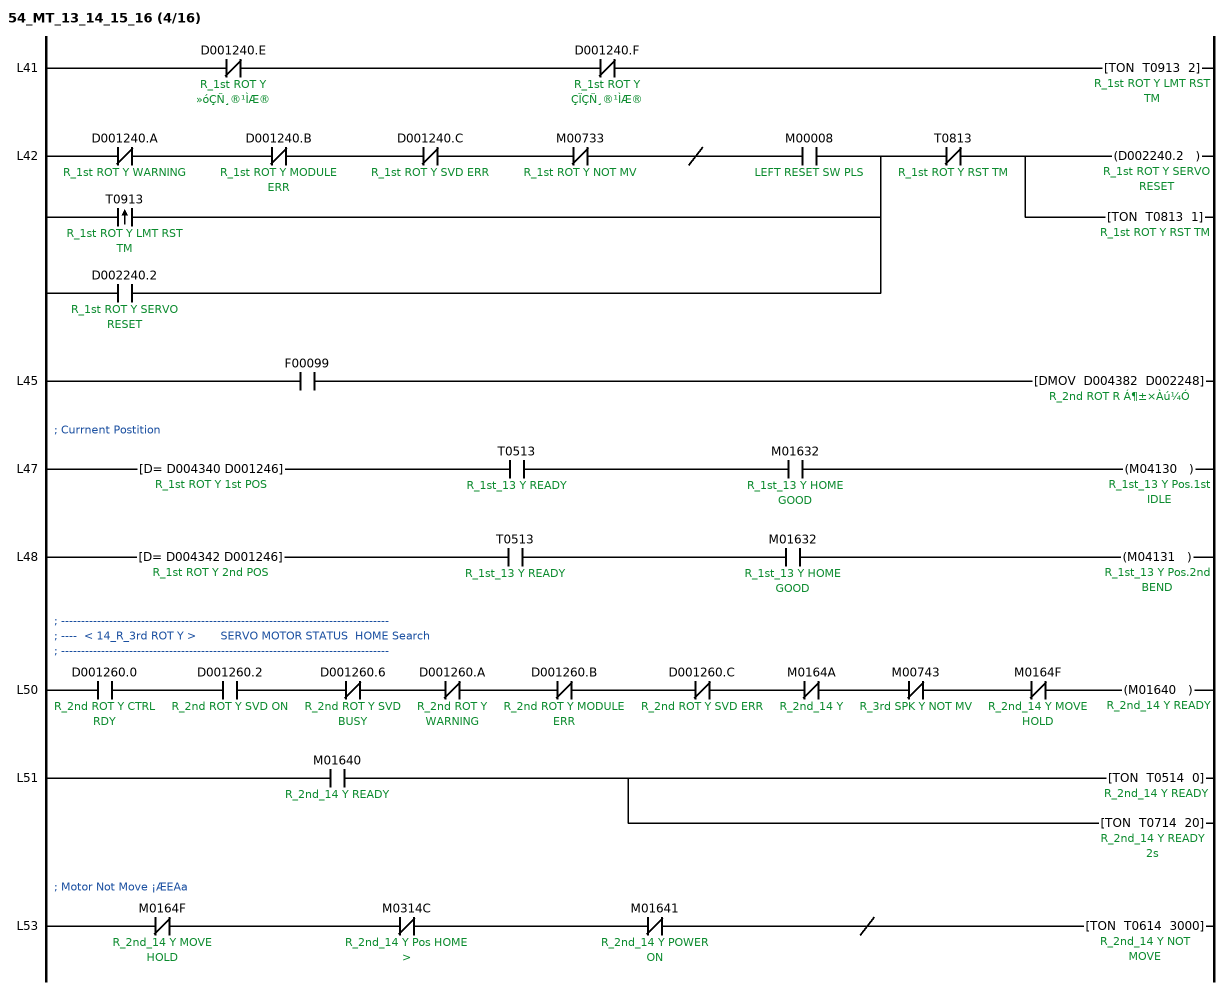
[picture p312: 54_MT_13_14_15_16 rungs L41-L53]
; L41
LOAD NOT  D001240.E	// R_1st ROT Y »óÇÑ¸®¹ÌÆ®
AND NOT   D001240.F	// R_1st ROT Y ÇÏÇÑ¸®¹ÌÆ®
TON       T0913 2	// R_1st ROT Y LMT RST TM
; L42
LOAD NOT  D001240.A	// R_1st ROT Y WARNING
AND NOT   D001240.B	// R_1st ROT Y MODULE ERR
AND NOT   D001240.C	// R_1st ROT Y SVD ERR
AND NOT   M00733	// R_1st ROT Y NOT MV
NOT
AND       M00008	// LEFT RESET SW PLS
ORP       T0913	// R_1st ROT Y LMT RST TM
OR        D002240.2	// R_1st ROT Y SERVO RESET
AND NOT   T0813	// R_1st ROT Y RST TM
OUT       D002240.2	// R_1st ROT Y SERVO RESET
TON       T0813 1	// R_1st ROT Y RST TM
; L45
LOAD      F00099
DMOV      D004382 D002248	// R_2nd ROT R Á¶±×Àú¼Ó
// Currnent Postition
; L47
LOADD=    D004340 D001246	// R_1st ROT Y 1st POS
AND       T0513	// R_1st_13 Y READY
AND       M01632	// R_1st_13 Y HOME GOOD
OUT       M04130	// R_1st_13 Y Pos.1st IDLE
; L48
LOADD=    D004342 D001246	// R_1st ROT Y 2nd POS
AND       T0513	// R_1st_13 Y READY
AND       M01632	// R_1st_13 Y HOME GOOD
OUT       M04131	// R_1st_13 Y Pos.2nd BEND
// ----------------------------------------------------------------------------------
// 
// ----  < 14_R_3rd ROT Y >       SERVO MOTOR STATUS  HOME Search
// 
// ----------------------------------------------------------------------------------
; L50
LOAD      D001260.0	// R_2nd ROT Y CTRL RDY
AND       D001260.2	// R_2nd ROT Y SVD ON
AND NOT   D001260.6	// R_2nd ROT Y SVD BUSY
AND NOT   D001260.A	// R_2nd ROT Y WARNING
AND NOT   D001260.B	// R_2nd ROT Y MODULE ERR
AND NOT   D001260.C	// R_2nd ROT Y SVD ERR
AND NOT   M0164A	// R_2nd_14 Y
AND NOT   M00743	// R_3rd SPK Y NOT MV
AND NOT   M0164F	// R_2nd_14 Y MOVE HOLD
OUT       M01640	// R_2nd_14 Y READY
; L51
LOAD      M01640	// R_2nd_14 Y READY
TON       T0514 0	// R_2nd_14 Y READY
TON       T0714 20	// R_2nd_14 Y READY 2s
; L53
LOAD NOT  M0164F	// R_2nd_14 Y MOVE HOLD
AND NOT   M0314C	// R_2nd_14 Y Pos HOME >
AND NOT   M01641	// R_2nd_14 Y POWER ON
NOT
TON       T0614 3000	// R_2nd_14 Y NOT MOVE
// output comment: Motor Not Move ¡ÆEAa

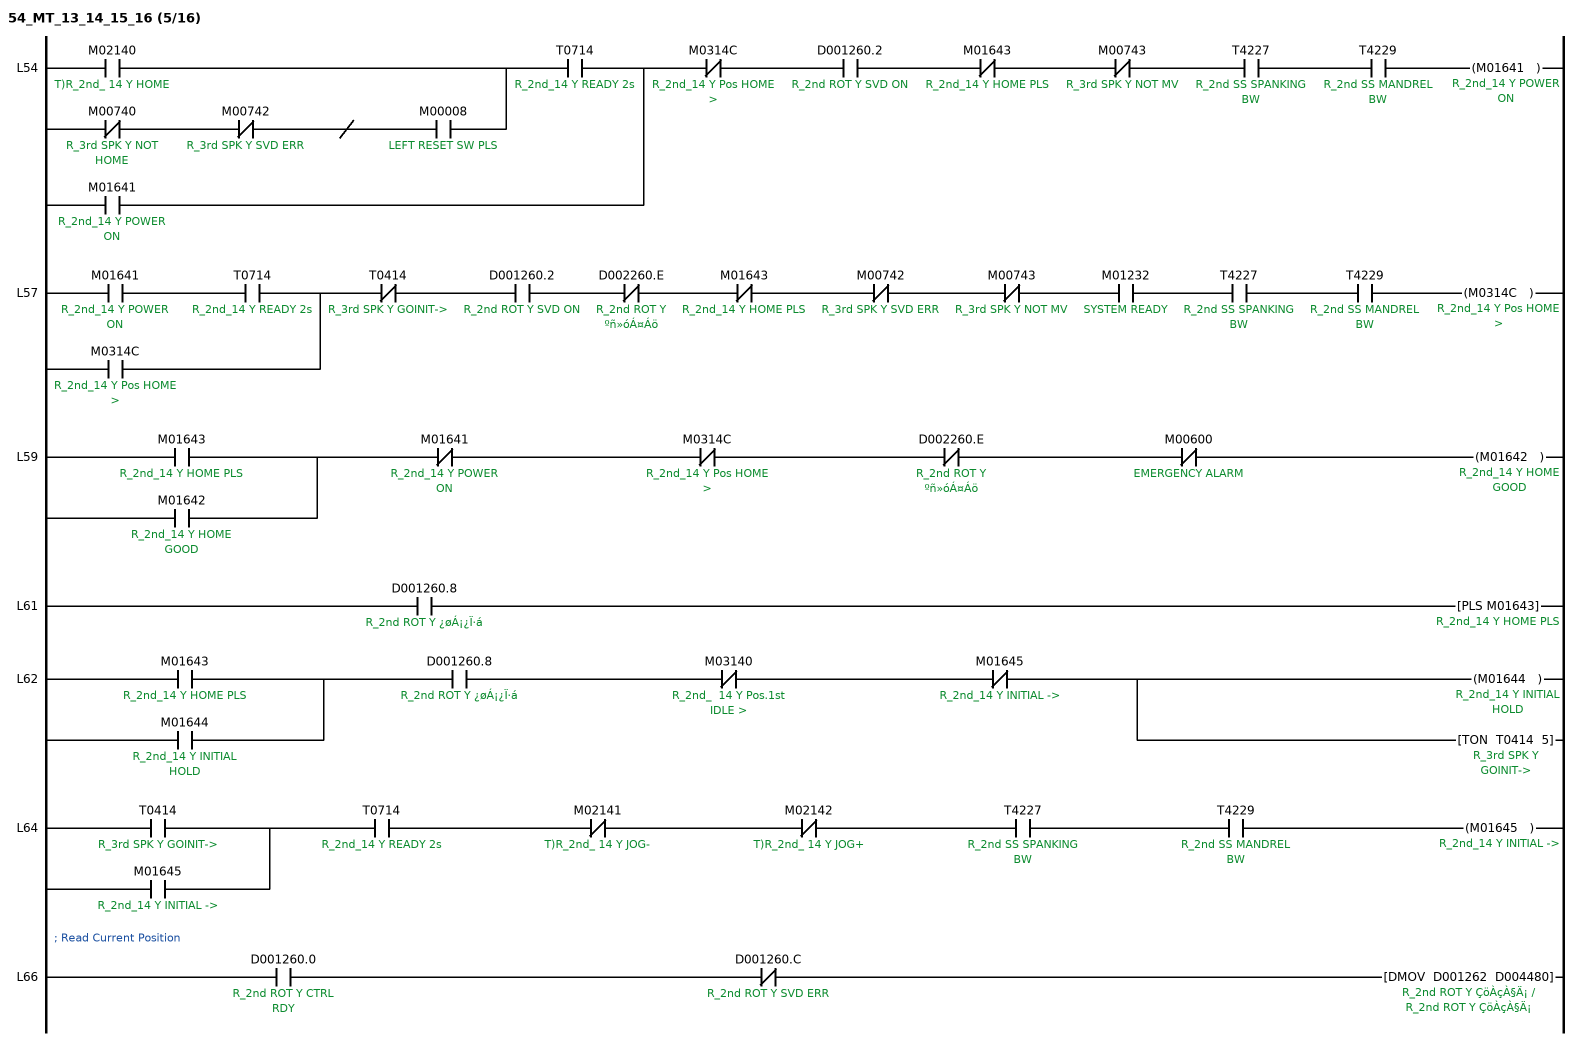
; L54
LOAD      M02140	// T)R_2nd_ 14 Y HOME
LOAD NOT  M00740	// R_3rd SPK Y NOT HOME
AND NOT   M00742	// R_3rd SPK Y SVD ERR
NOT
AND       M00008	// LEFT RESET SW PLS
OR LOAD
AND       T0714	// R_2nd_14 Y READY 2s
OR        M01641	// R_2nd_14 Y POWER ON
AND NOT   M0314C	// R_2nd_14 Y Pos HOME >
AND       D001260.2	// R_2nd ROT Y SVD ON
AND NOT   M01643	// R_2nd_14 Y HOME PLS
AND NOT   M00743	// R_3rd SPK Y NOT MV
AND       T4227	// R_2nd SS SPANKING BW
AND       T4229	// R_2nd SS MANDREL BW
OUT       M01641	// R_2nd_14 Y POWER ON
; L57
LOAD      M01641	// R_2nd_14 Y POWER ON
AND       T0714	// R_2nd_14 Y READY 2s
OR        M0314C	// R_2nd_14 Y Pos HOME >
AND NOT   T0414	// R_3rd SPK Y GOINIT->
AND       D001260.2	// R_2nd ROT Y SVD ON
AND NOT   D002260.E	// R_2nd ROT Y ºñ»óÁ¤Áö
AND NOT   M01643	// R_2nd_14 Y HOME PLS
AND NOT   M00742	// R_3rd SPK Y SVD ERR
AND NOT   M00743	// R_3rd SPK Y NOT MV
AND       M01232	// SYSTEM READY
AND       T4227	// R_2nd SS SPANKING BW
AND       T4229	// R_2nd SS MANDREL BW
OUT       M0314C	// R_2nd_14 Y Pos HOME >
; L59
LOAD      M01643	// R_2nd_14 Y HOME PLS
OR        M01642	// R_2nd_14 Y HOME GOOD
AND NOT   M01641	// R_2nd_14 Y POWER ON
AND NOT   M0314C	// R_2nd_14 Y Pos HOME >
AND NOT   D002260.E	// R_2nd ROT Y ºñ»óÁ¤Áö
AND NOT   M00600	// EMERGENCY ALARM
OUT       M01642	// R_2nd_14 Y HOME GOOD
; L61
LOAD      D001260.8	// R_2nd ROT Y ¿øÁ¡¿Ï·á
OUTP      M01643	// R_2nd_14 Y HOME PLS
; L62
LOAD      M01643	// R_2nd_14 Y HOME PLS
OR        M01644	// R_2nd_14 Y INITIAL HOLD
AND       D001260.8	// R_2nd ROT Y ¿øÁ¡¿Ï·á
AND NOT   M03140	// R_2nd_  14 Y Pos.1st IDLE >
AND NOT   M01645	// R_2nd_14 Y INITIAL ->
OUT       M01644	// R_2nd_14 Y INITIAL HOLD
TON       T0414 5	// R_3rd SPK Y GOINIT->
; L64
LOAD      T0414	// R_3rd SPK Y GOINIT->
OR        M01645	// R_2nd_14 Y INITIAL ->
AND       T0714	// R_2nd_14 Y READY 2s
AND NOT   M02141	// T)R_2nd_ 14 Y JOG-
AND NOT   M02142	// T)R_2nd_ 14 Y JOG+
AND       T4227	// R_2nd SS SPANKING BW
AND       T4229	// R_2nd SS MANDREL BW
OUT       M01645	// R_2nd_14 Y INITIAL ->
; L66
LOAD      D001260.0	// R_2nd ROT Y CTRL RDY
AND NOT   D001260.C	// R_2nd ROT Y SVD ERR
DMOV      D001262 D004480	// R_2nd ROT Y ÇöÀçÀ§Ä¡ / R_2nd ROT Y ÇöÀçÀ§Ä¡
// output comment: Read Current Position

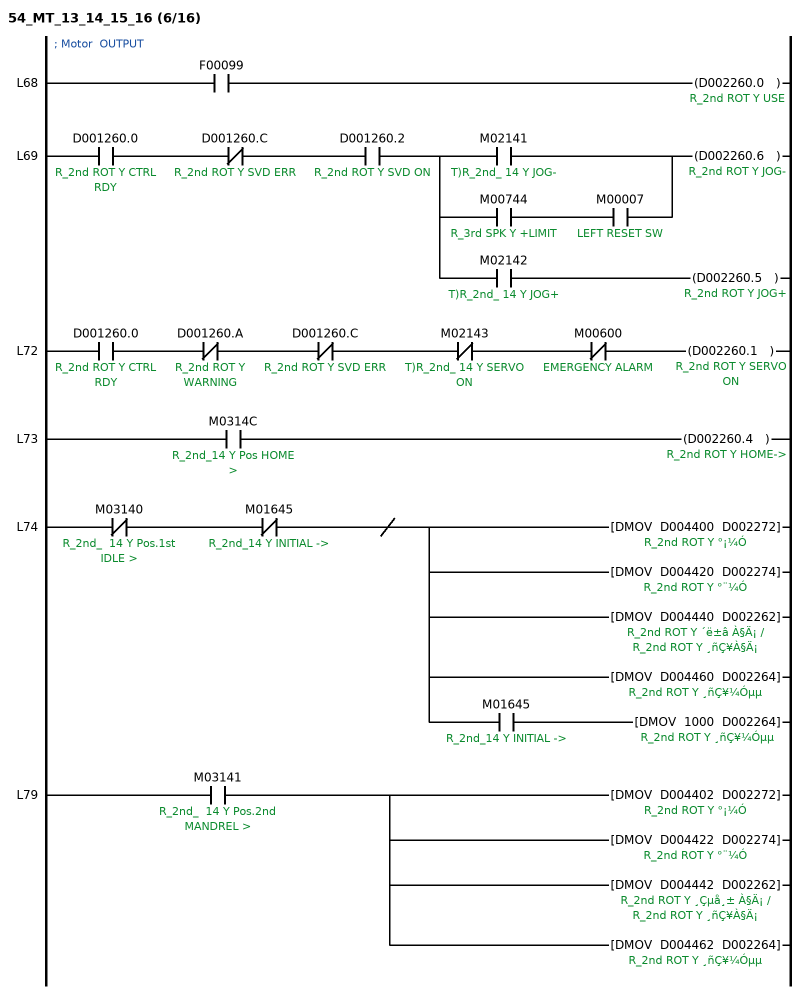
//  Motor  OUTPUT
; L68
LOAD      F00099
OUT       D002260.0	// R_2nd ROT Y USE
; L69
LOAD      D001260.0	// R_2nd ROT Y CTRL RDY
AND NOT   D001260.C	// R_2nd ROT Y SVD ERR
AND       D001260.2	// R_2nd ROT Y SVD ON
MPUSH
LOAD      M02141	// T)R_2nd_ 14 Y JOG-
LOAD      M00744	// R_3rd SPK Y +LIMIT
AND       M00007	// LEFT RESET SW
OR LOAD
AND LOAD
OUT       D002260.6	// R_2nd ROT Y JOG-
MPOP
AND       M02142	// T)R_2nd_ 14 Y JOG+
OUT       D002260.5	// R_2nd ROT Y JOG+
; L72
LOAD      D001260.0	// R_2nd ROT Y CTRL RDY
AND NOT   D001260.A	// R_2nd ROT Y WARNING
AND NOT   D001260.C	// R_2nd ROT Y SVD ERR
AND NOT   M02143	// T)R_2nd_ 14 Y SERVO ON
AND NOT   M00600	// EMERGENCY ALARM
OUT       D002260.1	// R_2nd ROT Y SERVO ON
; L73
LOAD      M0314C	// R_2nd_14 Y Pos HOME >
OUT       D002260.4	// R_2nd ROT Y HOME->
; L74
LOAD NOT  M03140	// R_2nd_  14 Y Pos.1st IDLE >
AND NOT   M01645	// R_2nd_14 Y INITIAL ->
NOT
DMOV      D004400 D002272	// R_2nd ROT Y °¡¼Ó
DMOV      D004420 D002274	// R_2nd ROT Y °¨¼Ó
DMOV      D004440 D002262	// R_2nd ROT Y ´ë±â À§Ä¡ / R_2nd ROT Y ¸ñÇ¥À§Ä¡
DMOV      D004460 D002264	// R_2nd ROT Y ¸ñÇ¥¼Óµµ
AND       M01645	// R_2nd_14 Y INITIAL ->
DMOV      1000 D002264	// R_2nd ROT Y ¸ñÇ¥¼Óµµ
; L79
LOAD      M03141	// R_2nd_  14 Y Pos.2nd MANDREL >
DMOV      D004402 D002272	// R_2nd ROT Y °¡¼Ó
DMOV      D004422 D002274	// R_2nd ROT Y °¨¼Ó
DMOV      D004442 D002262	// R_2nd ROT Y ¸Çµå¸± À§Ä¡ / R_2nd ROT Y ¸ñÇ¥À§Ä¡
DMOV      D004462 D002264	// R_2nd ROT Y ¸ñÇ¥¼Óµµ

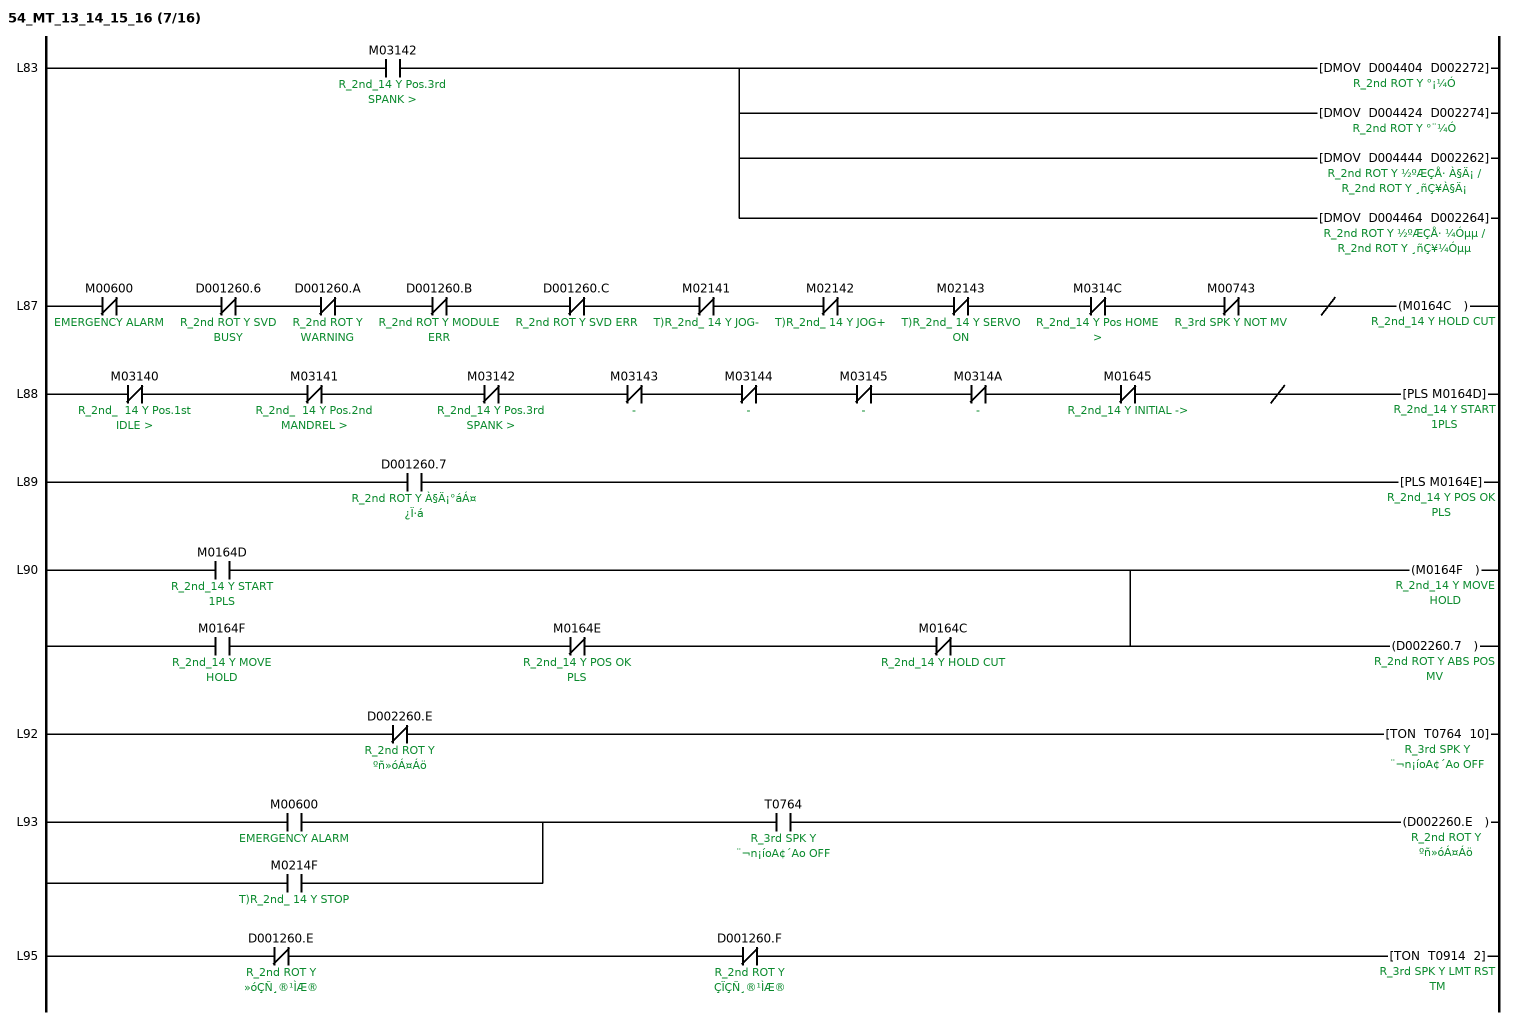
; L83
LOAD      M03142	// R_2nd_14 Y Pos.3rd SPANK >
DMOV      D004404 D002272	// R_2nd ROT Y °¡¼Ó
DMOV      D004424 D002274	// R_2nd ROT Y °¨¼Ó
DMOV      D004444 D002262	// R_2nd ROT Y ½ºÆÇÅ· À§Ä¡ / R_2nd ROT Y ¸ñÇ¥À§Ä¡
DMOV      D004464 D002264	// R_2nd ROT Y ½ºÆÇÅ· ¼Óµµ / R_2nd ROT Y ¸ñÇ¥¼Óµµ
; L87
LOAD NOT  M00600	// EMERGENCY ALARM
AND NOT   D001260.6	// R_2nd ROT Y SVD BUSY
AND NOT   D001260.A	// R_2nd ROT Y WARNING
AND NOT   D001260.B	// R_2nd ROT Y MODULE ERR
AND NOT   D001260.C	// R_2nd ROT Y SVD ERR
AND NOT   M02141	// T)R_2nd_ 14 Y JOG-
AND NOT   M02142	// T)R_2nd_ 14 Y JOG+
AND NOT   M02143	// T)R_2nd_ 14 Y SERVO ON
AND NOT   M0314C	// R_2nd_14 Y Pos HOME >
AND NOT   M00743	// R_3rd SPK Y NOT MV
NOT
OUT       M0164C	// R_2nd_14 Y HOLD CUT
; L88
LOAD NOT  M03140	// R_2nd_  14 Y Pos.1st IDLE >
AND NOT   M03141	// R_2nd_  14 Y Pos.2nd MANDREL >
AND NOT   M03142	// R_2nd_14 Y Pos.3rd SPANK >
AND NOT   M03143	// -
AND NOT   M03144	// -
AND NOT   M03145	// -
AND NOT   M0314A	// -
AND NOT   M01645	// R_2nd_14 Y INITIAL ->
NOT
OUTP      M0164D	// R_2nd_14 Y START 1PLS
; L89
LOAD      D001260.7	// R_2nd ROT Y À§Ä¡°áÁ¤ ¿Ï·á
OUTP      M0164E	// R_2nd_14 Y POS OK PLS
; L90
LOAD      M0164D	// R_2nd_14 Y START 1PLS
LOAD      M0164F	// R_2nd_14 Y MOVE HOLD
AND NOT   M0164E	// R_2nd_14 Y POS OK PLS
AND NOT   M0164C	// R_2nd_14 Y HOLD CUT
OR LOAD
OUT       M0164F	// R_2nd_14 Y MOVE HOLD
OUT       D002260.7	// R_2nd ROT Y ABS POS MV
; L92
LOAD NOT  D002260.E	// R_2nd ROT Y ºñ»óÁ¤Áö
TON       T0764 10	// R_3rd SPK Y ¨¬n¡íoA¢´Ao OFF
; L93
LOAD      M00600	// EMERGENCY ALARM
OR        M0214F	// T)R_2nd_ 14 Y STOP
AND       T0764	// R_3rd SPK Y ¨¬n¡íoA¢´Ao OFF
OUT       D002260.E	// R_2nd ROT Y ºñ»óÁ¤Áö
; L95
LOAD NOT  D001260.E	// R_2nd ROT Y »óÇÑ¸®¹ÌÆ®
AND NOT   D001260.F	// R_2nd ROT Y ÇÏÇÑ¸®¹ÌÆ®
TON       T0914 2	// R_3rd SPK Y LMT RST TM

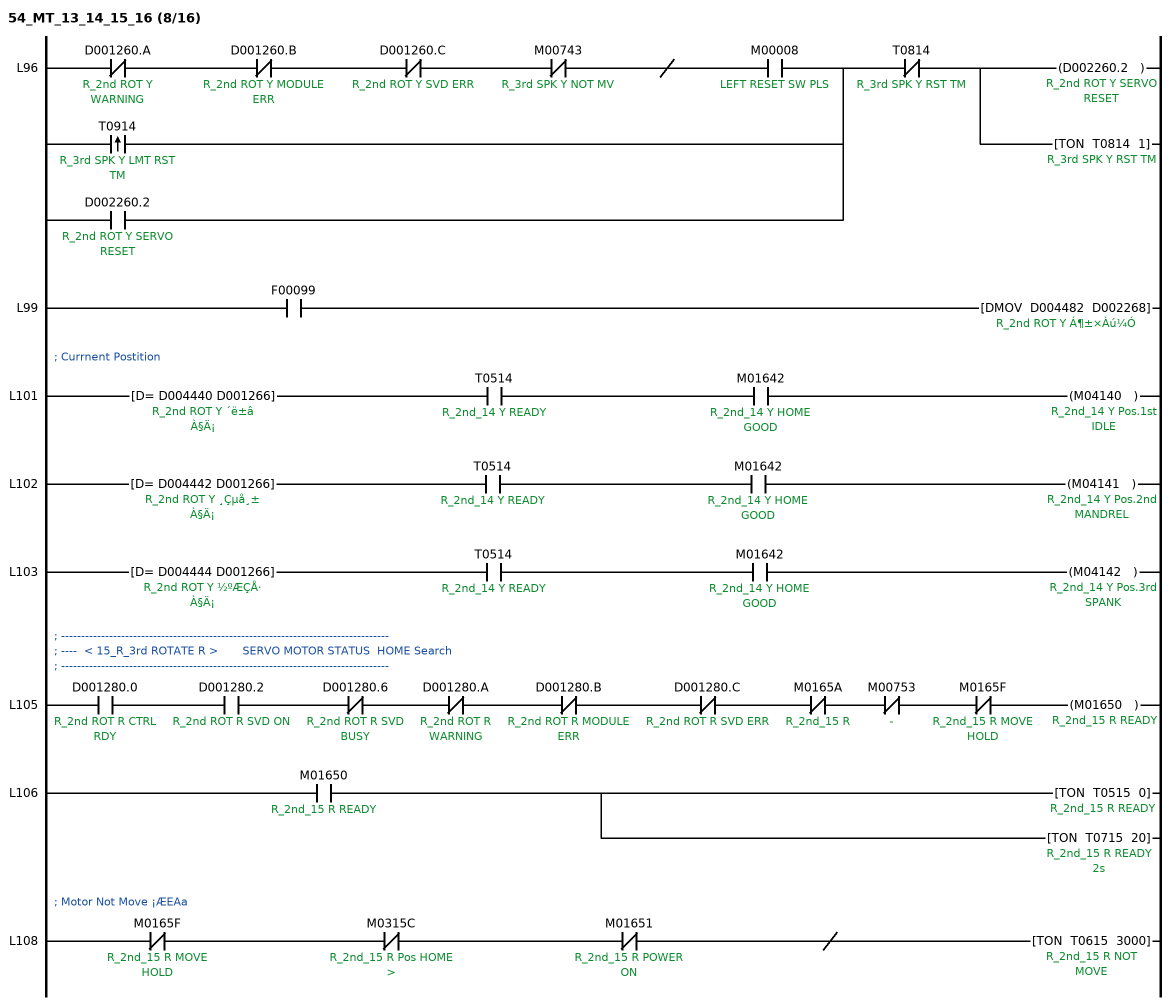
; L96
LOAD NOT  D001260.A	// R_2nd ROT Y WARNING
AND NOT   D001260.B	// R_2nd ROT Y MODULE ERR
AND NOT   D001260.C	// R_2nd ROT Y SVD ERR
AND NOT   M00743	// R_3rd SPK Y NOT MV
NOT
AND       M00008	// LEFT RESET SW PLS
ORP       T0914	// R_3rd SPK Y LMT RST TM
OR        D002260.2	// R_2nd ROT Y SERVO RESET
AND NOT   T0814	// R_3rd SPK Y RST TM
OUT       D002260.2	// R_2nd ROT Y SERVO RESET
TON       T0814 1	// R_3rd SPK Y RST TM
; L99
LOAD      F00099
DMOV      D004482 D002268	// R_2nd ROT Y Á¶±×Àú¼Ó
// Currnent Postition
; L101
LOADD=    D004440 D001266	// R_2nd ROT Y ´ë±â À§Ä¡
AND       T0514	// R_2nd_14 Y READY
AND       M01642	// R_2nd_14 Y HOME GOOD
OUT       M04140	// R_2nd_14 Y Pos.1st IDLE
; L102
LOADD=    D004442 D001266	// R_2nd ROT Y ¸Çµå¸± À§Ä¡
AND       T0514	// R_2nd_14 Y READY
AND       M01642	// R_2nd_14 Y HOME GOOD
OUT       M04141	// R_2nd_14 Y Pos.2nd MANDREL
; L103
LOADD=    D004444 D001266	// R_2nd ROT Y ½ºÆÇÅ· À§Ä¡
AND       T0514	// R_2nd_14 Y READY
AND       M01642	// R_2nd_14 Y HOME GOOD
OUT       M04142	// R_2nd_14 Y Pos.3rd SPANK
// ----------------------------------------------------------------------------------
// 
// ----  < 15_R_3rd ROTATE R >       SERVO MOTOR STATUS  HOME Search
// 
// ----------------------------------------------------------------------------------
; L105
LOAD      D001280.0	// R_2nd ROT R CTRL RDY
AND       D001280.2	// R_2nd ROT R SVD ON
AND NOT   D001280.6	// R_2nd ROT R SVD BUSY
AND NOT   D001280.A	// R_2nd ROT R WARNING
AND NOT   D001280.B	// R_2nd ROT R MODULE ERR
AND NOT   D001280.C	// R_2nd ROT R SVD ERR
AND NOT   M0165A	// R_2nd_15 R
AND NOT   M00753	// -
AND NOT   M0165F	// R_2nd_15 R MOVE HOLD
OUT       M01650	// R_2nd_15 R READY
; L106
LOAD      M01650	// R_2nd_15 R READY
TON       T0515 0	// R_2nd_15 R READY
TON       T0715 20	// R_2nd_15 R READY 2s
; L108
LOAD NOT  M0165F	// R_2nd_15 R MOVE HOLD
AND NOT   M0315C	// R_2nd_15 R Pos HOME >
AND NOT   M01651	// R_2nd_15 R POWER ON
NOT
TON       T0615 3000	// R_2nd_15 R NOT MOVE
// output comment: Motor Not Move ¡ÆEAa

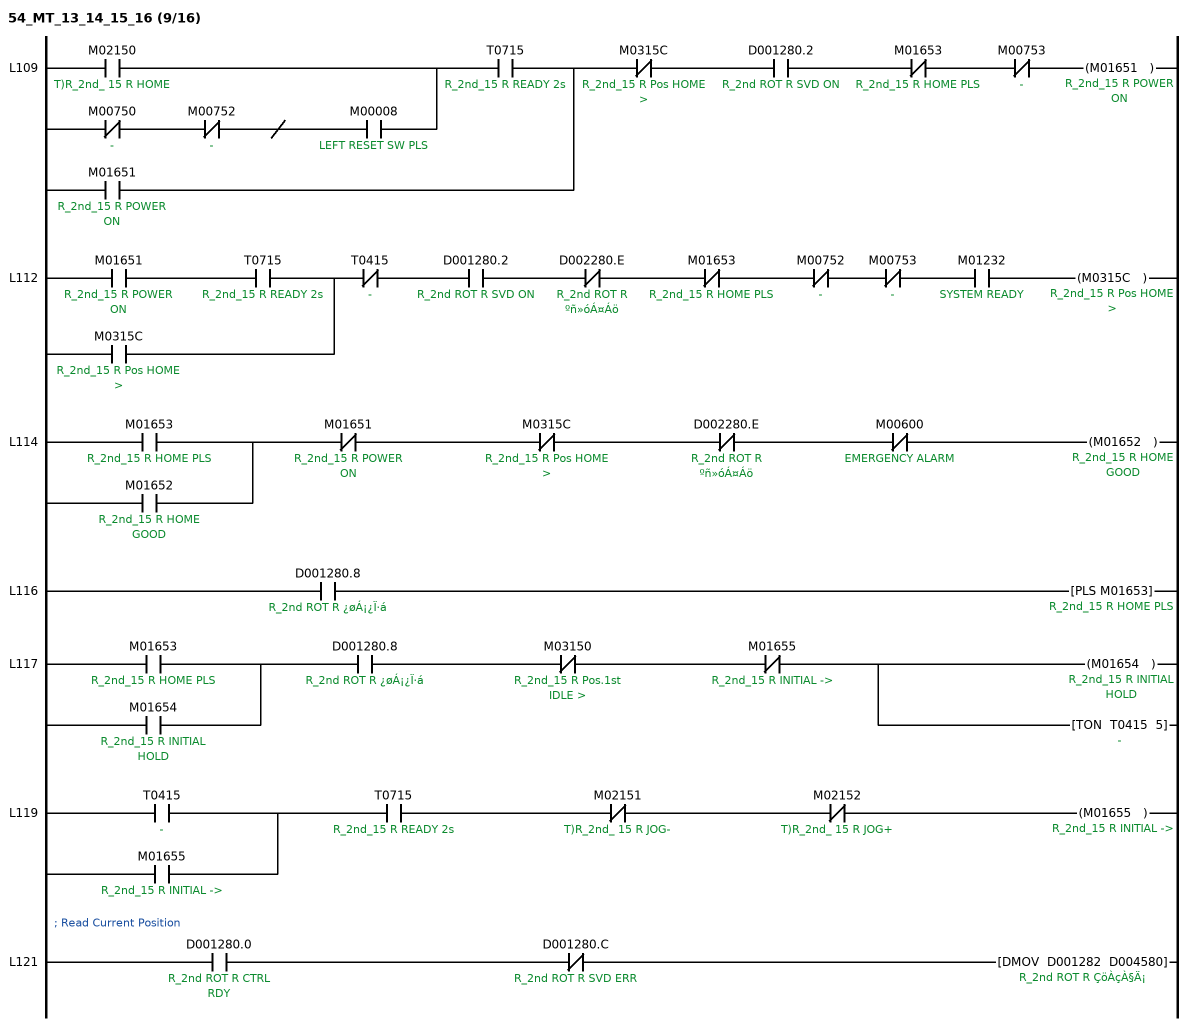
; L109
LOAD      M02150	// T)R_2nd_ 15 R HOME
LOAD NOT  M00750	// -
AND NOT   M00752	// -
NOT
AND       M00008	// LEFT RESET SW PLS
OR LOAD
AND       T0715	// R_2nd_15 R READY 2s
OR        M01651	// R_2nd_15 R POWER ON
AND NOT   M0315C	// R_2nd_15 R Pos HOME >
AND       D001280.2	// R_2nd ROT R SVD ON
AND NOT   M01653	// R_2nd_15 R HOME PLS
AND NOT   M00753	// -
OUT       M01651	// R_2nd_15 R POWER ON
; L112
LOAD      M01651	// R_2nd_15 R POWER ON
AND       T0715	// R_2nd_15 R READY 2s
OR        M0315C	// R_2nd_15 R Pos HOME >
AND NOT   T0415	// -
AND       D001280.2	// R_2nd ROT R SVD ON
AND NOT   D002280.E	// R_2nd ROT R ºñ»óÁ¤Áö
AND NOT   M01653	// R_2nd_15 R HOME PLS
AND NOT   M00752	// -
AND NOT   M00753	// -
AND       M01232	// SYSTEM READY
OUT       M0315C	// R_2nd_15 R Pos HOME >
; L114
LOAD      M01653	// R_2nd_15 R HOME PLS
OR        M01652	// R_2nd_15 R HOME GOOD
AND NOT   M01651	// R_2nd_15 R POWER ON
AND NOT   M0315C	// R_2nd_15 R Pos HOME >
AND NOT   D002280.E	// R_2nd ROT R ºñ»óÁ¤Áö
AND NOT   M00600	// EMERGENCY ALARM
OUT       M01652	// R_2nd_15 R HOME GOOD
; L116
LOAD      D001280.8	// R_2nd ROT R ¿øÁ¡¿Ï·á
OUTP      M01653	// R_2nd_15 R HOME PLS
; L117
LOAD      M01653	// R_2nd_15 R HOME PLS
OR        M01654	// R_2nd_15 R INITIAL HOLD
AND       D001280.8	// R_2nd ROT R ¿øÁ¡¿Ï·á
AND NOT   M03150	// R_2nd_15 R Pos.1st IDLE >
AND NOT   M01655	// R_2nd_15 R INITIAL ->
OUT       M01654	// R_2nd_15 R INITIAL HOLD
TON       T0415 5	// -
; L119
LOAD      T0415	// -
OR        M01655	// R_2nd_15 R INITIAL ->
AND       T0715	// R_2nd_15 R READY 2s
AND NOT   M02151	// T)R_2nd_ 15 R JOG-
AND NOT   M02152	// T)R_2nd_ 15 R JOG+
OUT       M01655	// R_2nd_15 R INITIAL ->
; L121
LOAD      D001280.0	// R_2nd ROT R CTRL RDY
AND NOT   D001280.C	// R_2nd ROT R SVD ERR
DMOV      D001282 D004580	// R_2nd ROT R ÇöÀçÀ§Ä¡
// output comment: Read Current Position

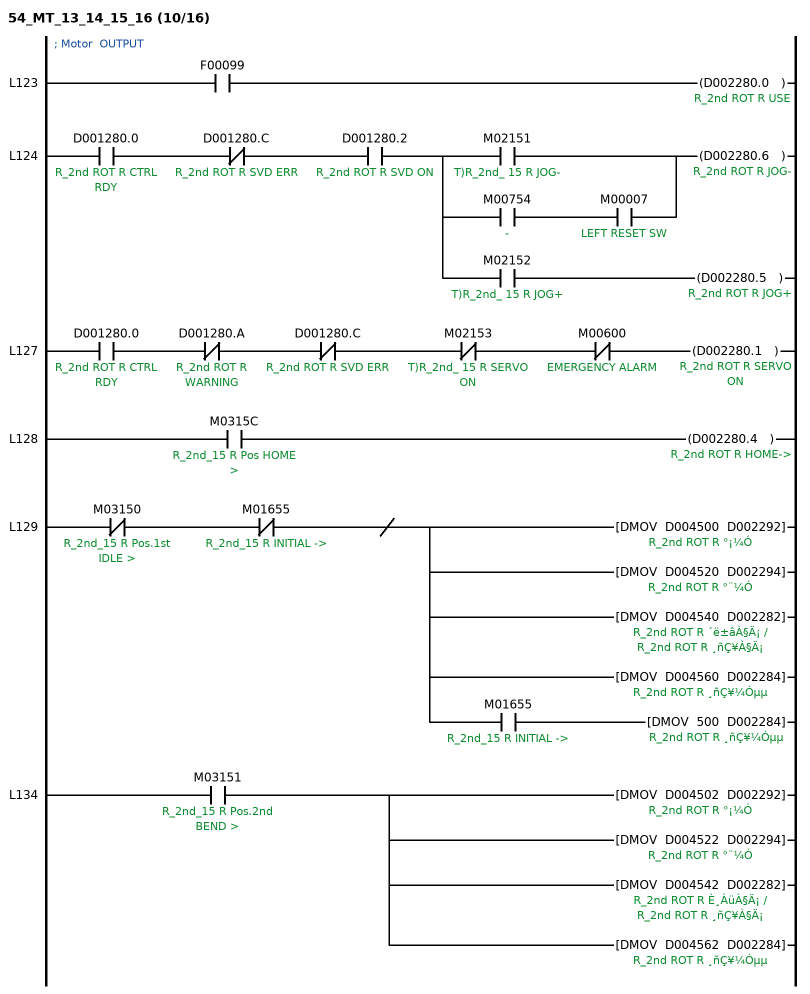
//  Motor  OUTPUT
; L123
LOAD      F00099
OUT       D002280.0	// R_2nd ROT R USE
; L124
LOAD      D001280.0	// R_2nd ROT R CTRL RDY
AND NOT   D001280.C	// R_2nd ROT R SVD ERR
AND       D001280.2	// R_2nd ROT R SVD ON
MPUSH
LOAD      M02151	// T)R_2nd_ 15 R JOG-
LOAD      M00754	// -
AND       M00007	// LEFT RESET SW
OR LOAD
AND LOAD
OUT       D002280.6	// R_2nd ROT R JOG-
MPOP
AND       M02152	// T)R_2nd_ 15 R JOG+
OUT       D002280.5	// R_2nd ROT R JOG+
; L127
LOAD      D001280.0	// R_2nd ROT R CTRL RDY
AND NOT   D001280.A	// R_2nd ROT R WARNING
AND NOT   D001280.C	// R_2nd ROT R SVD ERR
AND NOT   M02153	// T)R_2nd_ 15 R SERVO ON
AND NOT   M00600	// EMERGENCY ALARM
OUT       D002280.1	// R_2nd ROT R SERVO ON
; L128
LOAD      M0315C	// R_2nd_15 R Pos HOME >
OUT       D002280.4	// R_2nd ROT R HOME->
; L129
LOAD NOT  M03150	// R_2nd_15 R Pos.1st IDLE >
AND NOT   M01655	// R_2nd_15 R INITIAL ->
NOT
DMOV      D004500 D002292	// R_2nd ROT R °¡¼Ó
DMOV      D004520 D002294	// R_2nd ROT R °¨¼Ó
DMOV      D004540 D002282	// R_2nd ROT R ´ë±âÀ§Ä¡ / R_2nd ROT R ¸ñÇ¥À§Ä¡
DMOV      D004560 D002284	// R_2nd ROT R ¸ñÇ¥¼Óµµ
AND       M01655	// R_2nd_15 R INITIAL ->
DMOV      500 D002284	// R_2nd ROT R ¸ñÇ¥¼Óµµ
; L134
LOAD      M03151	// R_2nd_15 R Pos.2nd BEND >
DMOV      D004502 D002292	// R_2nd ROT R °¡¼Ó
DMOV      D004522 D002294	// R_2nd ROT R °¨¼Ó
DMOV      D004542 D002282	// R_2nd ROT R È¸ÀüÀ§Ä¡ / R_2nd ROT R ¸ñÇ¥À§Ä¡
DMOV      D004562 D002284	// R_2nd ROT R ¸ñÇ¥¼Óµµ

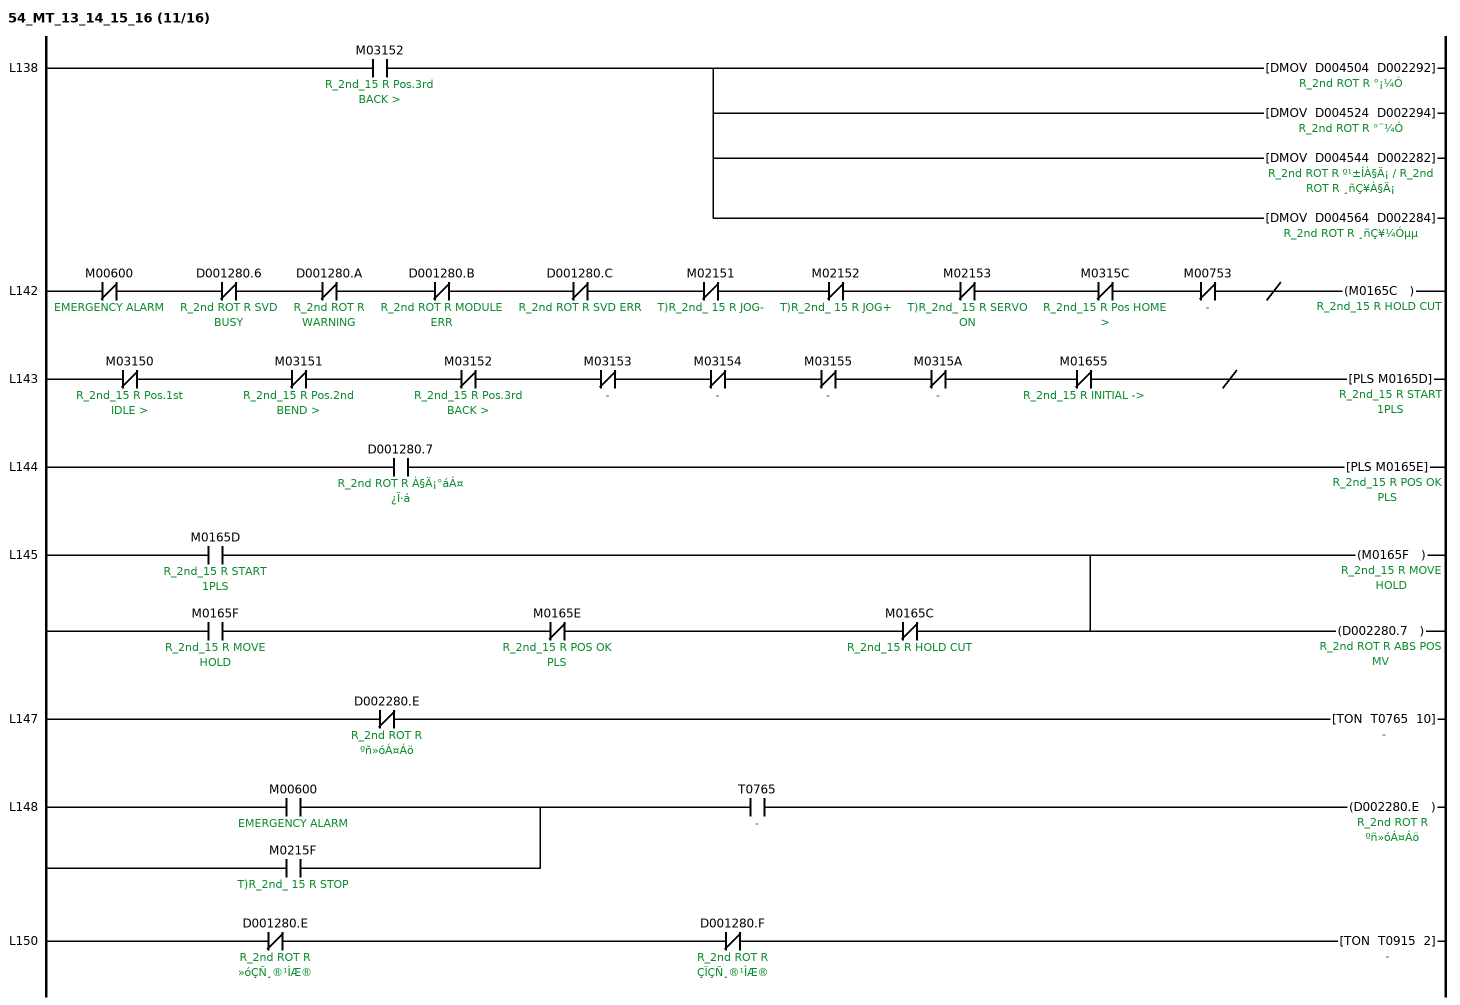
; L138
LOAD      M03152	// R_2nd_15 R Pos.3rd BACK >
DMOV      D004504 D002292	// R_2nd ROT R °¡¼Ó
DMOV      D004524 D002294	// R_2nd ROT R °¨¼Ó
DMOV      D004544 D002282	// R_2nd ROT R º¹±ÍÀ§Ä¡ / R_2nd ROT R ¸ñÇ¥À§Ä¡
DMOV      D004564 D002284	// R_2nd ROT R ¸ñÇ¥¼Óµµ
; L142
LOAD NOT  M00600	// EMERGENCY ALARM
AND NOT   D001280.6	// R_2nd ROT R SVD BUSY
AND NOT   D001280.A	// R_2nd ROT R WARNING
AND NOT   D001280.B	// R_2nd ROT R MODULE ERR
AND NOT   D001280.C	// R_2nd ROT R SVD ERR
AND NOT   M02151	// T)R_2nd_ 15 R JOG-
AND NOT   M02152	// T)R_2nd_ 15 R JOG+
AND NOT   M02153	// T)R_2nd_ 15 R SERVO ON
AND NOT   M0315C	// R_2nd_15 R Pos HOME >
AND NOT   M00753	// -
NOT
OUT       M0165C	// R_2nd_15 R HOLD CUT
; L143
LOAD NOT  M03150	// R_2nd_15 R Pos.1st IDLE >
AND NOT   M03151	// R_2nd_15 R Pos.2nd BEND >
AND NOT   M03152	// R_2nd_15 R Pos.3rd BACK >
AND NOT   M03153	// -
AND NOT   M03154	// -
AND NOT   M03155	// -
AND NOT   M0315A	// -
AND NOT   M01655	// R_2nd_15 R INITIAL ->
NOT
OUTP      M0165D	// R_2nd_15 R START 1PLS
; L144
LOAD      D001280.7	// R_2nd ROT R À§Ä¡°áÁ¤ ¿Ï·á
OUTP      M0165E	// R_2nd_15 R POS OK PLS
; L145
LOAD      M0165D	// R_2nd_15 R START 1PLS
LOAD      M0165F	// R_2nd_15 R MOVE HOLD
AND NOT   M0165E	// R_2nd_15 R POS OK PLS
AND NOT   M0165C	// R_2nd_15 R HOLD CUT
OR LOAD
OUT       M0165F	// R_2nd_15 R MOVE HOLD
OUT       D002280.7	// R_2nd ROT R ABS POS MV
; L147
LOAD NOT  D002280.E	// R_2nd ROT R ºñ»óÁ¤Áö
TON       T0765 10	// -
; L148
LOAD      M00600	// EMERGENCY ALARM
OR        M0215F	// T)R_2nd_ 15 R STOP
AND       T0765	// -
OUT       D002280.E	// R_2nd ROT R ºñ»óÁ¤Áö
; L150
LOAD NOT  D001280.E	// R_2nd ROT R »óÇÑ¸®¹ÌÆ®
AND NOT   D001280.F	// R_2nd ROT R ÇÏÇÑ¸®¹ÌÆ®
TON       T0915 2	// -

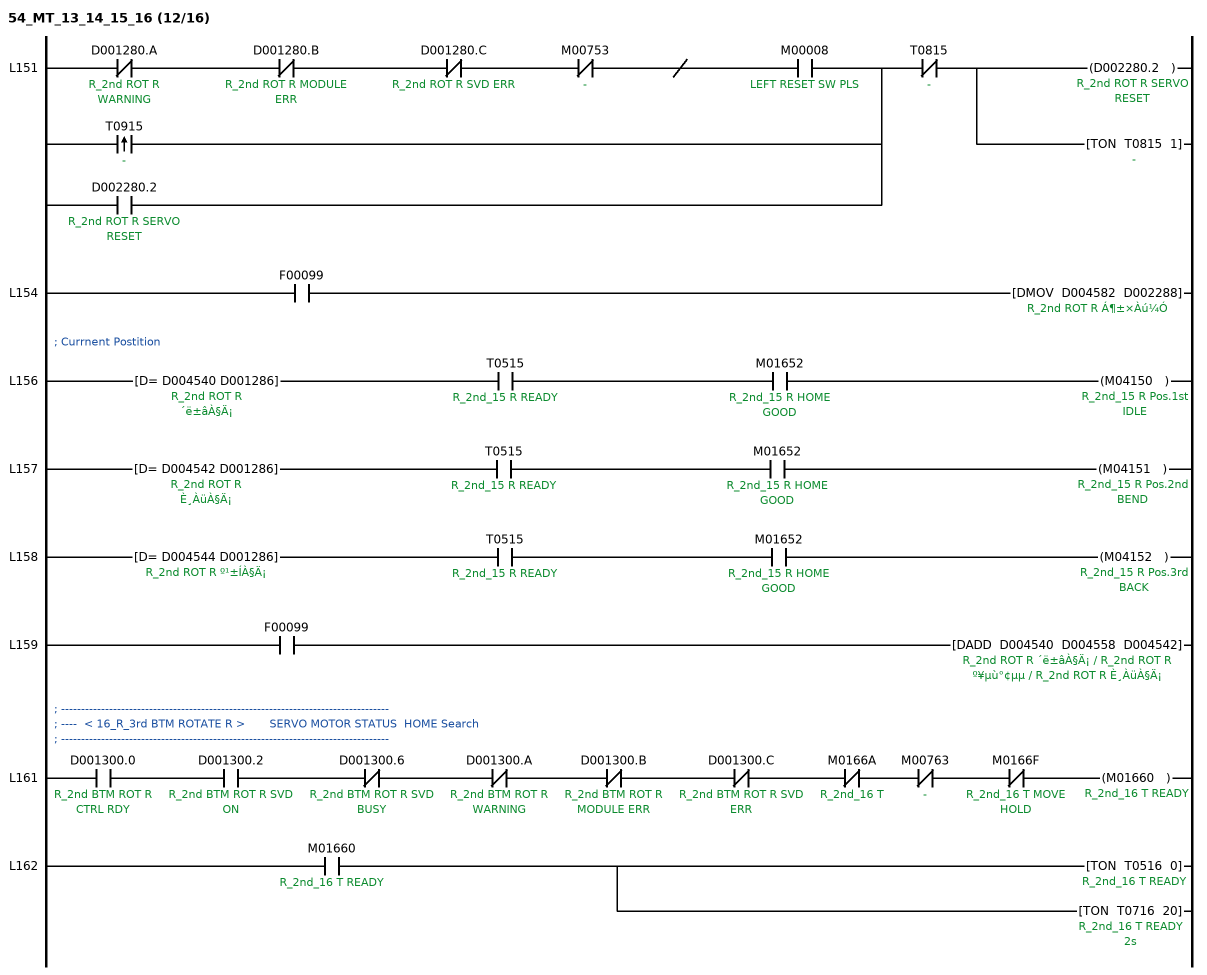
; L151
LOAD NOT  D001280.A	// R_2nd ROT R WARNING
AND NOT   D001280.B	// R_2nd ROT R MODULE ERR
AND NOT   D001280.C	// R_2nd ROT R SVD ERR
AND NOT   M00753	// -
NOT
AND       M00008	// LEFT RESET SW PLS
ORP       T0915	// -
OR        D002280.2	// R_2nd ROT R SERVO RESET
AND NOT   T0815	// -
OUT       D002280.2	// R_2nd ROT R SERVO RESET
TON       T0815 1	// -
; L154
LOAD      F00099
DMOV      D004582 D002288	// R_2nd ROT R Á¶±×Àú¼Ó
// Currnent Postition
; L156
LOADD=    D004540 D001286	// R_2nd ROT R ´ë±âÀ§Ä¡
AND       T0515	// R_2nd_15 R READY
AND       M01652	// R_2nd_15 R HOME GOOD
OUT       M04150	// R_2nd_15 R Pos.1st IDLE
; L157
LOADD=    D004542 D001286	// R_2nd ROT R È¸ÀüÀ§Ä¡
AND       T0515	// R_2nd_15 R READY
AND       M01652	// R_2nd_15 R HOME GOOD
OUT       M04151	// R_2nd_15 R Pos.2nd BEND
; L158
LOADD=    D004544 D001286	// R_2nd ROT R º¹±ÍÀ§Ä¡
AND       T0515	// R_2nd_15 R READY
AND       M01652	// R_2nd_15 R HOME GOOD
OUT       M04152	// R_2nd_15 R Pos.3rd BACK
; L159
LOAD      F00099
DADD      D004540 D004558 D004542	// R_2nd ROT R ´ë±âÀ§Ä¡ / R_2nd ROT R º¥µù°¢µµ / R_2nd ROT R È¸ÀüÀ§Ä¡
// ----------------------------------------------------------------------------------
// 
// ----  < 16_R_3rd BTM ROTATE R >       SERVO MOTOR STATUS  HOME Search
// 
// ----------------------------------------------------------------------------------
; L161
LOAD      D001300.0	// R_2nd BTM ROT R CTRL RDY
AND       D001300.2	// R_2nd BTM ROT R SVD ON
AND NOT   D001300.6	// R_2nd BTM ROT R SVD BUSY
AND NOT   D001300.A	// R_2nd BTM ROT R WARNING
AND NOT   D001300.B	// R_2nd BTM ROT R MODULE ERR
AND NOT   D001300.C	// R_2nd BTM ROT R SVD ERR
AND NOT   M0166A	// R_2nd_16 T
AND NOT   M00763	// -
AND NOT   M0166F	// R_2nd_16 T MOVE HOLD
OUT       M01660	// R_2nd_16 T READY
; L162
LOAD      M01660	// R_2nd_16 T READY
TON       T0516 0	// R_2nd_16 T READY
TON       T0716 20	// R_2nd_16 T READY 2s

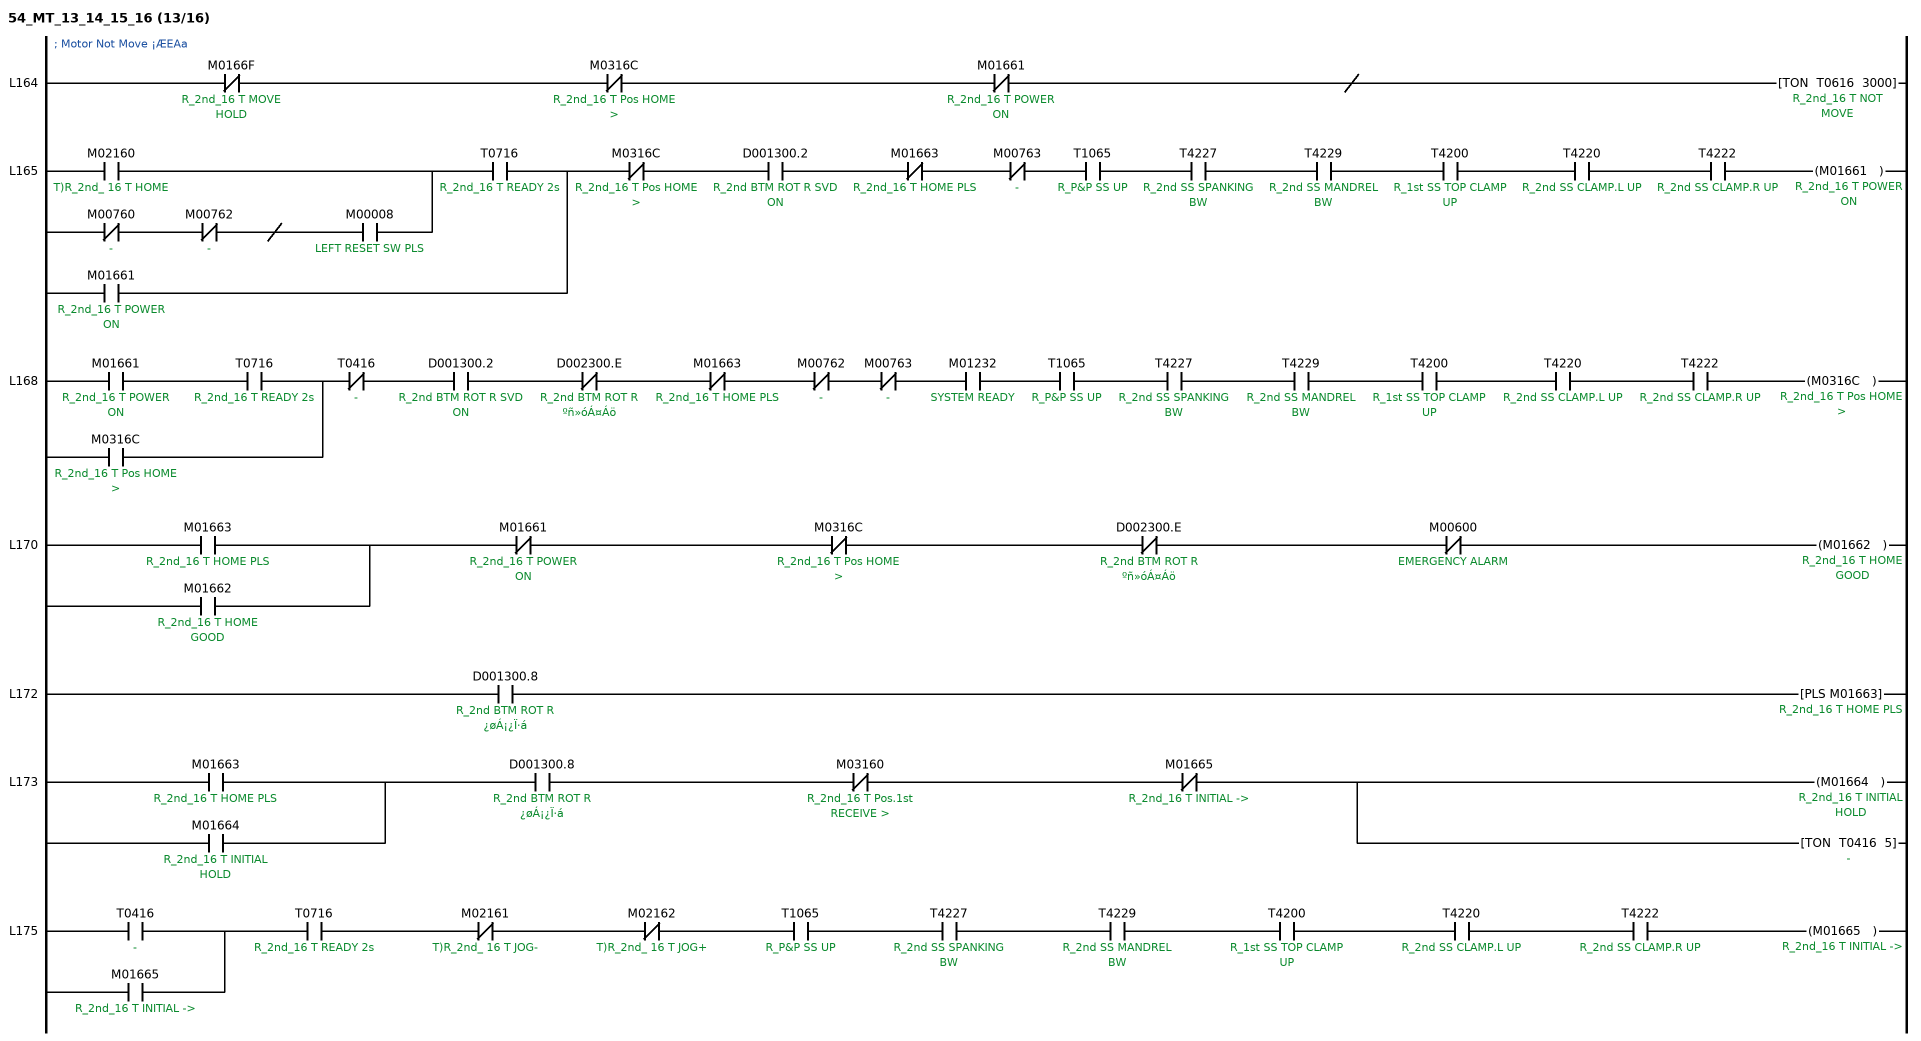
; L164
LOAD NOT  M0166F	// R_2nd_16 T MOVE HOLD
AND NOT   M0316C	// R_2nd_16 T Pos HOME >
AND NOT   M01661	// R_2nd_16 T POWER ON
NOT
TON       T0616 3000	// R_2nd_16 T NOT MOVE
// output comment: Motor Not Move ¡ÆEAa
; L165
LOAD      M02160	// T)R_2nd_ 16 T HOME
LOAD NOT  M00760	// -
AND NOT   M00762	// -
NOT
AND       M00008	// LEFT RESET SW PLS
OR LOAD
AND       T0716	// R_2nd_16 T READY 2s
OR        M01661	// R_2nd_16 T POWER ON
AND NOT   M0316C	// R_2nd_16 T Pos HOME >
AND       D001300.2	// R_2nd BTM ROT R SVD ON
AND NOT   M01663	// R_2nd_16 T HOME PLS
AND NOT   M00763	// -
AND       T1065	// R_P&P SS UP
AND       T4227	// R_2nd SS SPANKING BW
AND       T4229	// R_2nd SS MANDREL BW
AND       T4200	// R_1st SS TOP CLAMP UP
AND       T4220	// R_2nd SS CLAMP.L UP
AND       T4222	// R_2nd SS CLAMP.R UP
OUT       M01661	// R_2nd_16 T POWER ON
; L168
LOAD      M01661	// R_2nd_16 T POWER ON
AND       T0716	// R_2nd_16 T READY 2s
OR        M0316C	// R_2nd_16 T Pos HOME >
AND NOT   T0416	// -
AND       D001300.2	// R_2nd BTM ROT R SVD ON
AND NOT   D002300.E	// R_2nd BTM ROT R ºñ»óÁ¤Áö
AND NOT   M01663	// R_2nd_16 T HOME PLS
AND NOT   M00762	// -
AND NOT   M00763	// -
AND       M01232	// SYSTEM READY
AND       T1065	// R_P&P SS UP
AND       T4227	// R_2nd SS SPANKING BW
AND       T4229	// R_2nd SS MANDREL BW
AND       T4200	// R_1st SS TOP CLAMP UP
AND       T4220	// R_2nd SS CLAMP.L UP
AND       T4222	// R_2nd SS CLAMP.R UP
OUT       M0316C	// R_2nd_16 T Pos HOME >
; L170
LOAD      M01663	// R_2nd_16 T HOME PLS
OR        M01662	// R_2nd_16 T HOME GOOD
AND NOT   M01661	// R_2nd_16 T POWER ON
AND NOT   M0316C	// R_2nd_16 T Pos HOME >
AND NOT   D002300.E	// R_2nd BTM ROT R ºñ»óÁ¤Áö
AND NOT   M00600	// EMERGENCY ALARM
OUT       M01662	// R_2nd_16 T HOME GOOD
; L172
LOAD      D001300.8	// R_2nd BTM ROT R ¿øÁ¡¿Ï·á
OUTP      M01663	// R_2nd_16 T HOME PLS
; L173
LOAD      M01663	// R_2nd_16 T HOME PLS
OR        M01664	// R_2nd_16 T INITIAL HOLD
AND       D001300.8	// R_2nd BTM ROT R ¿øÁ¡¿Ï·á
AND NOT   M03160	// R_2nd_16 T Pos.1st RECEIVE >
AND NOT   M01665	// R_2nd_16 T INITIAL ->
OUT       M01664	// R_2nd_16 T INITIAL HOLD
TON       T0416 5	// -
; L175
LOAD      T0416	// -
OR        M01665	// R_2nd_16 T INITIAL ->
AND       T0716	// R_2nd_16 T READY 2s
AND NOT   M02161	// T)R_2nd_ 16 T JOG-
AND NOT   M02162	// T)R_2nd_ 16 T JOG+
AND       T1065	// R_P&P SS UP
AND       T4227	// R_2nd SS SPANKING BW
AND       T4229	// R_2nd SS MANDREL BW
AND       T4200	// R_1st SS TOP CLAMP UP
AND       T4220	// R_2nd SS CLAMP.L UP
AND       T4222	// R_2nd SS CLAMP.R UP
OUT       M01665	// R_2nd_16 T INITIAL ->

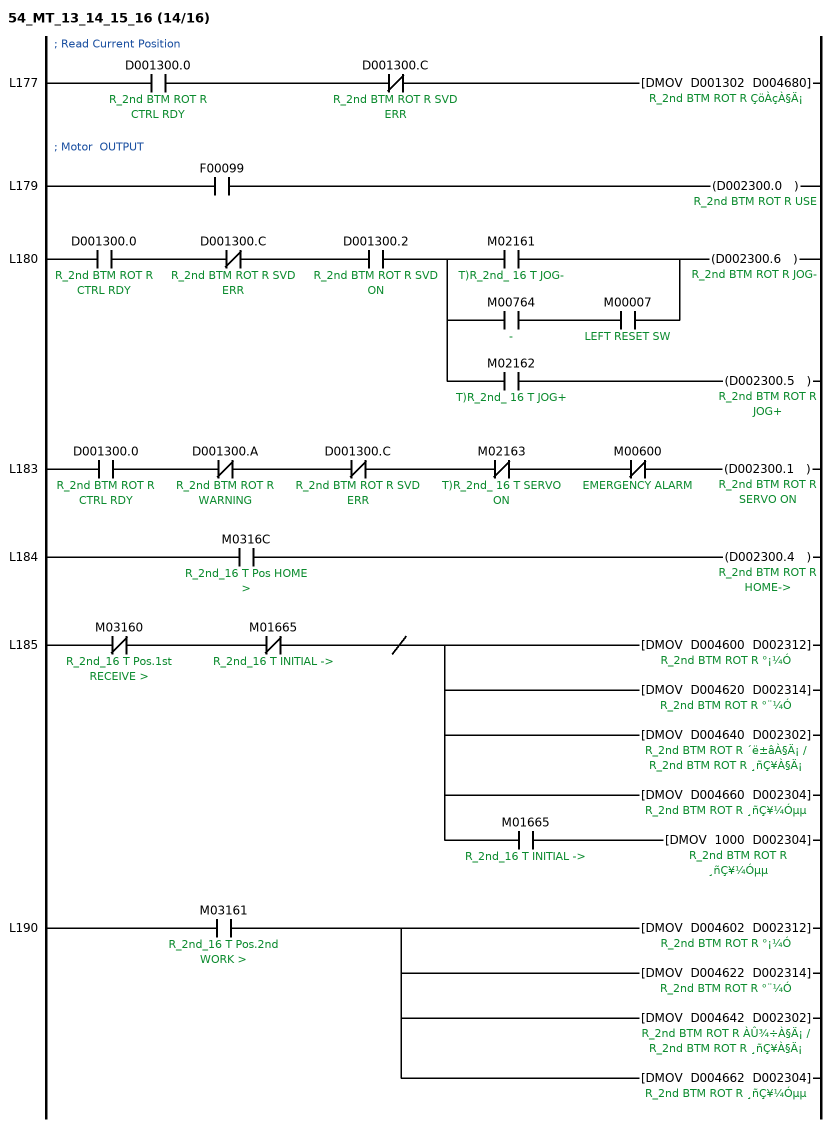
; L177
LOAD      D001300.0	// R_2nd BTM ROT R CTRL RDY
AND NOT   D001300.C	// R_2nd BTM ROT R SVD ERR
DMOV      D001302 D004680	// R_2nd BTM ROT R ÇöÀçÀ§Ä¡
// output comment: Read Current Position
//  Motor  OUTPUT
; L179
LOAD      F00099
OUT       D002300.0	// R_2nd BTM ROT R USE
; L180
LOAD      D001300.0	// R_2nd BTM ROT R CTRL RDY
AND NOT   D001300.C	// R_2nd BTM ROT R SVD ERR
AND       D001300.2	// R_2nd BTM ROT R SVD ON
MPUSH
LOAD      M02161	// T)R_2nd_ 16 T JOG-
LOAD      M00764	// -
AND       M00007	// LEFT RESET SW
OR LOAD
AND LOAD
OUT       D002300.6	// R_2nd BTM ROT R JOG-
MPOP
AND       M02162	// T)R_2nd_ 16 T JOG+
OUT       D002300.5	// R_2nd BTM ROT R JOG+
; L183
LOAD      D001300.0	// R_2nd BTM ROT R CTRL RDY
AND NOT   D001300.A	// R_2nd BTM ROT R WARNING
AND NOT   D001300.C	// R_2nd BTM ROT R SVD ERR
AND NOT   M02163	// T)R_2nd_ 16 T SERVO ON
AND NOT   M00600	// EMERGENCY ALARM
OUT       D002300.1	// R_2nd BTM ROT R SERVO ON
; L184
LOAD      M0316C	// R_2nd_16 T Pos HOME >
OUT       D002300.4	// R_2nd BTM ROT R HOME->
; L185
LOAD NOT  M03160	// R_2nd_16 T Pos.1st RECEIVE >
AND NOT   M01665	// R_2nd_16 T INITIAL ->
NOT
DMOV      D004600 D002312	// R_2nd BTM ROT R °¡¼Ó
DMOV      D004620 D002314	// R_2nd BTM ROT R °¨¼Ó
DMOV      D004640 D002302	// R_2nd BTM ROT R ´ë±âÀ§Ä¡ / R_2nd BTM ROT R ¸ñÇ¥À§Ä¡
DMOV      D004660 D002304	// R_2nd BTM ROT R ¸ñÇ¥¼Óµµ
AND       M01665	// R_2nd_16 T INITIAL ->
DMOV      1000 D002304	// R_2nd BTM ROT R ¸ñÇ¥¼Óµµ
; L190
LOAD      M03161	// R_2nd_16 T Pos.2nd WORK >
DMOV      D004602 D002312	// R_2nd BTM ROT R °¡¼Ó
DMOV      D004622 D002314	// R_2nd BTM ROT R °¨¼Ó
DMOV      D004642 D002302	// R_2nd BTM ROT R ÀÛ¾÷À§Ä¡ / R_2nd BTM ROT R ¸ñÇ¥À§Ä¡
DMOV      D004662 D002304	// R_2nd BTM ROT R ¸ñÇ¥¼Óµµ

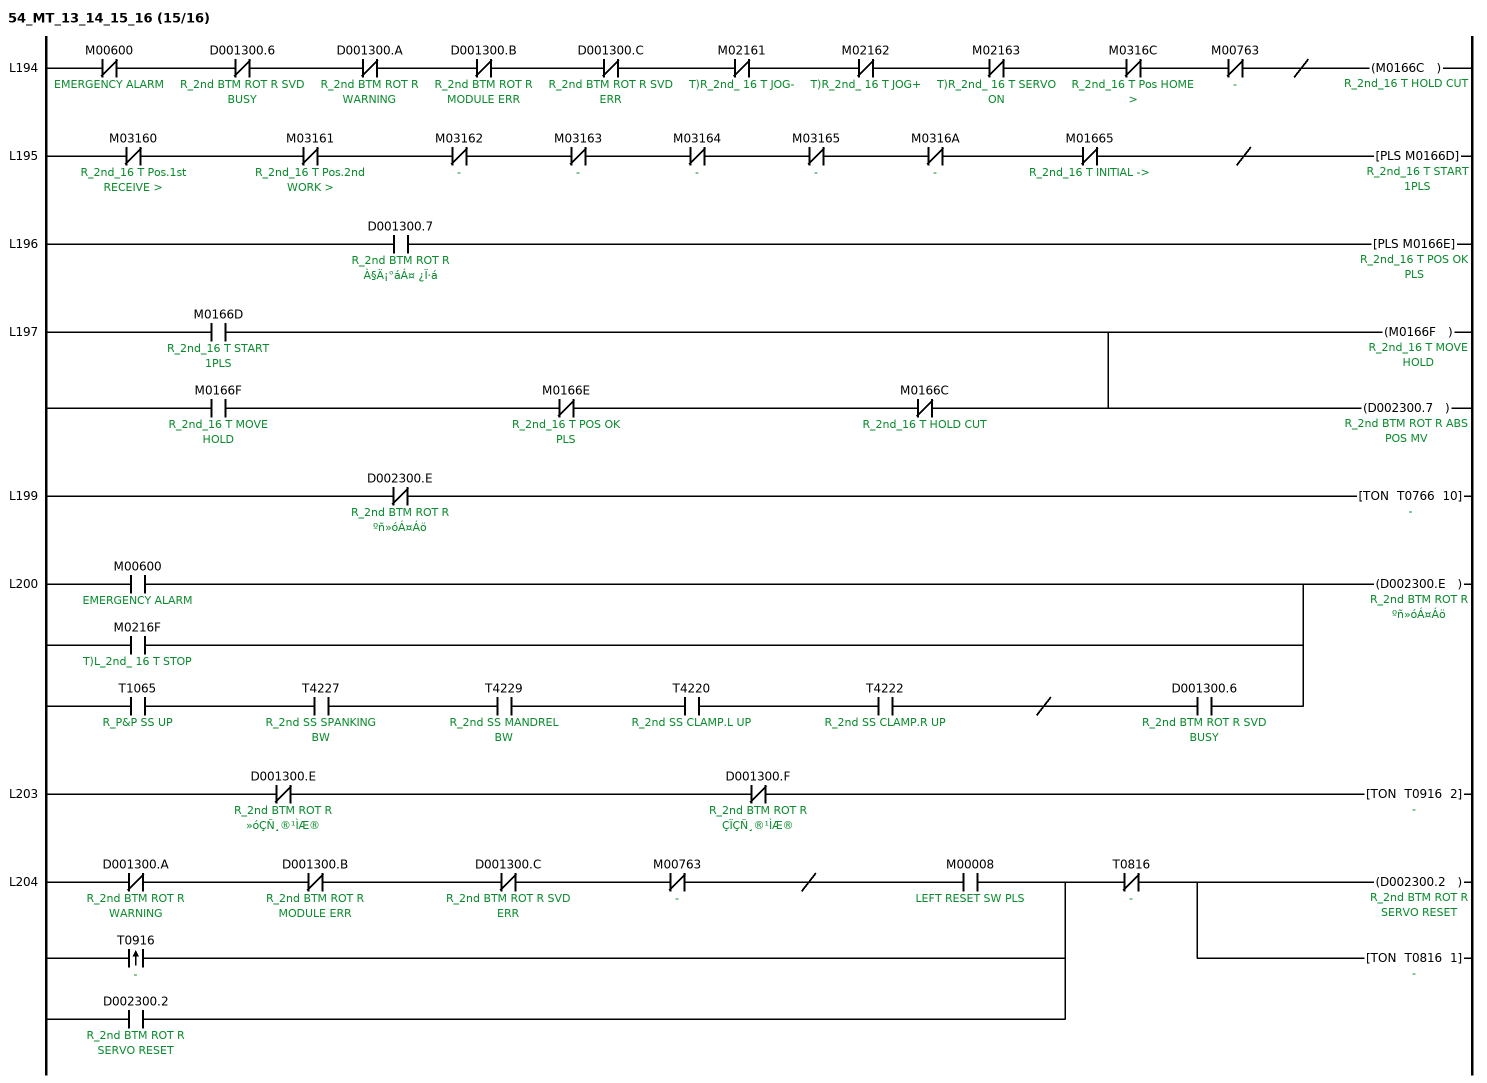
; L194
LOAD NOT  M00600	// EMERGENCY ALARM
AND NOT   D001300.6	// R_2nd BTM ROT R SVD BUSY
AND NOT   D001300.A	// R_2nd BTM ROT R WARNING
AND NOT   D001300.B	// R_2nd BTM ROT R MODULE ERR
AND NOT   D001300.C	// R_2nd BTM ROT R SVD ERR
AND NOT   M02161	// T)R_2nd_ 16 T JOG-
AND NOT   M02162	// T)R_2nd_ 16 T JOG+
AND NOT   M02163	// T)R_2nd_ 16 T SERVO ON
AND NOT   M0316C	// R_2nd_16 T Pos HOME >
AND NOT   M00763	// -
NOT
OUT       M0166C	// R_2nd_16 T HOLD CUT
; L195
LOAD NOT  M03160	// R_2nd_16 T Pos.1st RECEIVE >
AND NOT   M03161	// R_2nd_16 T Pos.2nd WORK >
AND NOT   M03162	// -
AND NOT   M03163	// -
AND NOT   M03164	// -
AND NOT   M03165	// -
AND NOT   M0316A	// -
AND NOT   M01665	// R_2nd_16 T INITIAL ->
NOT
OUTP      M0166D	// R_2nd_16 T START 1PLS
; L196
LOAD      D001300.7	// R_2nd BTM ROT R À§Ä¡°áÁ¤ ¿Ï·á
OUTP      M0166E	// R_2nd_16 T POS OK PLS
; L197
LOAD      M0166D	// R_2nd_16 T START 1PLS
LOAD      M0166F	// R_2nd_16 T MOVE HOLD
AND NOT   M0166E	// R_2nd_16 T POS OK PLS
AND NOT   M0166C	// R_2nd_16 T HOLD CUT
OR LOAD
OUT       M0166F	// R_2nd_16 T MOVE HOLD
OUT       D002300.7	// R_2nd BTM ROT R ABS POS MV
; L199
LOAD NOT  D002300.E	// R_2nd BTM ROT R ºñ»óÁ¤Áö
TON       T0766 10	// -
; L200
LOAD      M00600	// EMERGENCY ALARM
OR        M0216F	// T)L_2nd_ 16 T STOP
LOAD      T1065	// R_P&P SS UP
AND       T4227	// R_2nd SS SPANKING BW
AND       T4229	// R_2nd SS MANDREL BW
AND       T4220	// R_2nd SS CLAMP.L UP
AND       T4222	// R_2nd SS CLAMP.R UP
NOT
AND       D001300.6	// R_2nd BTM ROT R SVD BUSY
OR LOAD
OUT       D002300.E	// R_2nd BTM ROT R ºñ»óÁ¤Áö
; L203
LOAD NOT  D001300.E	// R_2nd BTM ROT R »óÇÑ¸®¹ÌÆ®
AND NOT   D001300.F	// R_2nd BTM ROT R ÇÏÇÑ¸®¹ÌÆ®
TON       T0916 2	// -
; L204
LOAD NOT  D001300.A	// R_2nd BTM ROT R WARNING
AND NOT   D001300.B	// R_2nd BTM ROT R MODULE ERR
AND NOT   D001300.C	// R_2nd BTM ROT R SVD ERR
AND NOT   M00763	// -
NOT
AND       M00008	// LEFT RESET SW PLS
ORP       T0916	// -
OR        D002300.2	// R_2nd BTM ROT R SERVO RESET
AND NOT   T0816	// -
OUT       D002300.2	// R_2nd BTM ROT R SERVO RESET
TON       T0816 1	// -

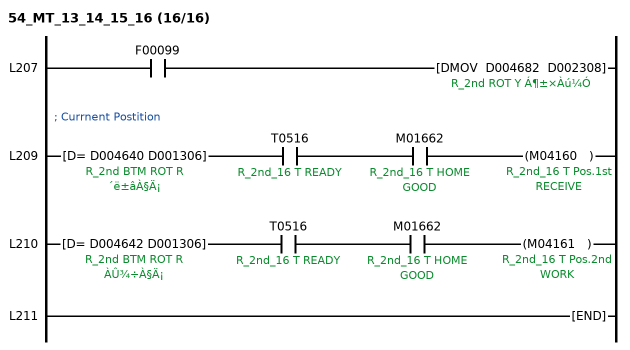
; L207
LOAD      F00099
DMOV      D004682 D002308	// R_2nd ROT Y Á¶±×Àú¼Ó
// Currnent Postition
; L209
LOADD=    D004640 D001306	// R_2nd BTM ROT R ´ë±âÀ§Ä¡
AND       T0516	// R_2nd_16 T READY
AND       M01662	// R_2nd_16 T HOME GOOD
OUT       M04160	// R_2nd_16 T Pos.1st RECEIVE
; L210
LOADD=    D004642 D001306	// R_2nd BTM ROT R ÀÛ¾÷À§Ä¡
AND       T0516	// R_2nd_16 T READY
AND       M01662	// R_2nd_16 T HOME GOOD
OUT       M04161	// R_2nd_16 T Pos.2nd WORK
; L211
END

PROGRAM 55_MT_17_18_19_20 (task: ½ºÄµ ÇÁ·Î±×·¥)

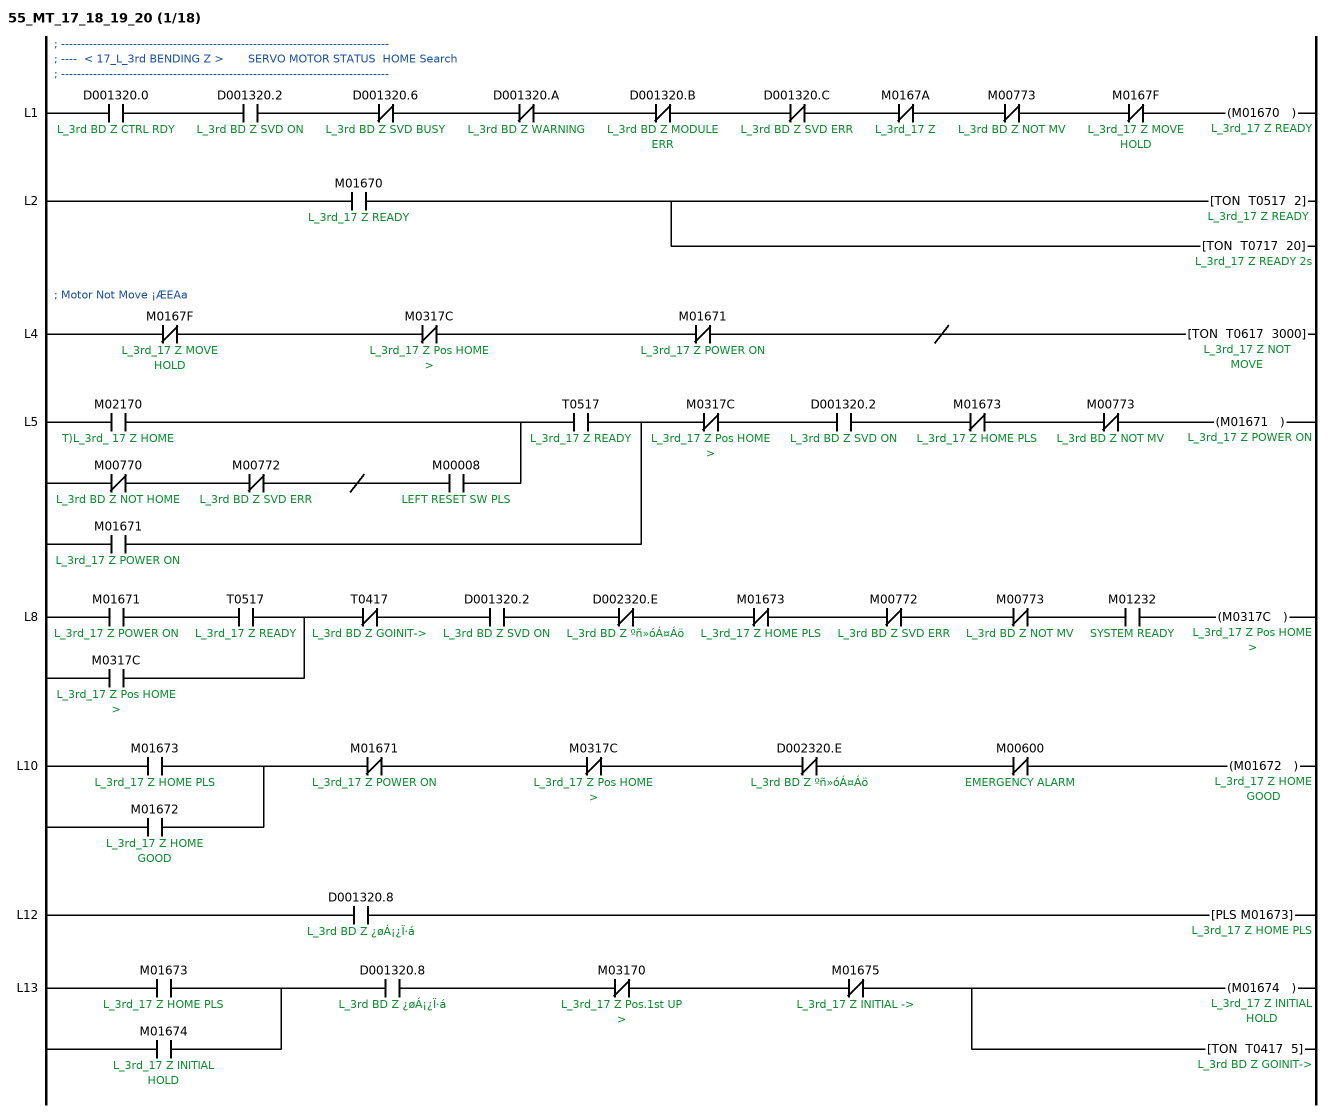
// ----------------------------------------------------------------------------------
// 
// ----  < 17_L_3rd BENDING Z >       SERVO MOTOR STATUS  HOME Search
// 
// ----------------------------------------------------------------------------------
; L1
LOAD      D001320.0	// L_3rd BD Z CTRL RDY
AND       D001320.2	// L_3rd BD Z SVD ON
AND NOT   D001320.6	// L_3rd BD Z SVD BUSY
AND NOT   D001320.A	// L_3rd BD Z WARNING
AND NOT   D001320.B	// L_3rd BD Z MODULE ERR
AND NOT   D001320.C	// L_3rd BD Z SVD ERR
AND NOT   M0167A	// L_3rd_17 Z
AND NOT   M00773	// L_3rd BD Z NOT MV
AND NOT   M0167F	// L_3rd_17 Z MOVE HOLD
OUT       M01670	// L_3rd_17 Z READY
; L2
LOAD      M01670	// L_3rd_17 Z READY
TON       T0517 2	// L_3rd_17 Z READY
TON       T0717 20	// L_3rd_17 Z READY 2s
; L4
LOAD NOT  M0167F	// L_3rd_17 Z MOVE HOLD
AND NOT   M0317C	// L_3rd_17 Z Pos HOME >
AND NOT   M01671	// L_3rd_17 Z POWER ON
NOT
TON       T0617 3000	// L_3rd_17 Z NOT MOVE
// output comment: Motor Not Move ¡ÆEAa
; L5
LOAD      M02170	// T)L_3rd_ 17 Z HOME
LOAD NOT  M00770	// L_3rd BD Z NOT HOME
AND NOT   M00772	// L_3rd BD Z SVD ERR
NOT
AND       M00008	// LEFT RESET SW PLS
OR LOAD
AND       T0517	// L_3rd_17 Z READY
OR        M01671	// L_3rd_17 Z POWER ON
AND NOT   M0317C	// L_3rd_17 Z Pos HOME >
AND       D001320.2	// L_3rd BD Z SVD ON
AND NOT   M01673	// L_3rd_17 Z HOME PLS
AND NOT   M00773	// L_3rd BD Z NOT MV
OUT       M01671	// L_3rd_17 Z POWER ON
; L8
LOAD      M01671	// L_3rd_17 Z POWER ON
AND       T0517	// L_3rd_17 Z READY
OR        M0317C	// L_3rd_17 Z Pos HOME >
AND NOT   T0417	// L_3rd BD Z GOINIT->
AND       D001320.2	// L_3rd BD Z SVD ON
AND NOT   D002320.E	// L_3rd BD Z ºñ»óÁ¤Áö
AND NOT   M01673	// L_3rd_17 Z HOME PLS
AND NOT   M00772	// L_3rd BD Z SVD ERR
AND NOT   M00773	// L_3rd BD Z NOT MV
AND       M01232	// SYSTEM READY
OUT       M0317C	// L_3rd_17 Z Pos HOME >
; L10
LOAD      M01673	// L_3rd_17 Z HOME PLS
OR        M01672	// L_3rd_17 Z HOME GOOD
AND NOT   M01671	// L_3rd_17 Z POWER ON
AND NOT   M0317C	// L_3rd_17 Z Pos HOME >
AND NOT   D002320.E	// L_3rd BD Z ºñ»óÁ¤Áö
AND NOT   M00600	// EMERGENCY ALARM
OUT       M01672	// L_3rd_17 Z HOME GOOD
; L12
LOAD      D001320.8	// L_3rd BD Z ¿øÁ¡¿Ï·á
OUTP      M01673	// L_3rd_17 Z HOME PLS
; L13
LOAD      M01673	// L_3rd_17 Z HOME PLS
OR        M01674	// L_3rd_17 Z INITIAL HOLD
AND       D001320.8	// L_3rd BD Z ¿øÁ¡¿Ï·á
AND NOT   M03170	// L_3rd_17 Z Pos.1st UP >
AND NOT   M01675	// L_3rd_17 Z INITIAL ->
OUT       M01674	// L_3rd_17 Z INITIAL HOLD
TON       T0417 5	// L_3rd BD Z GOINIT->

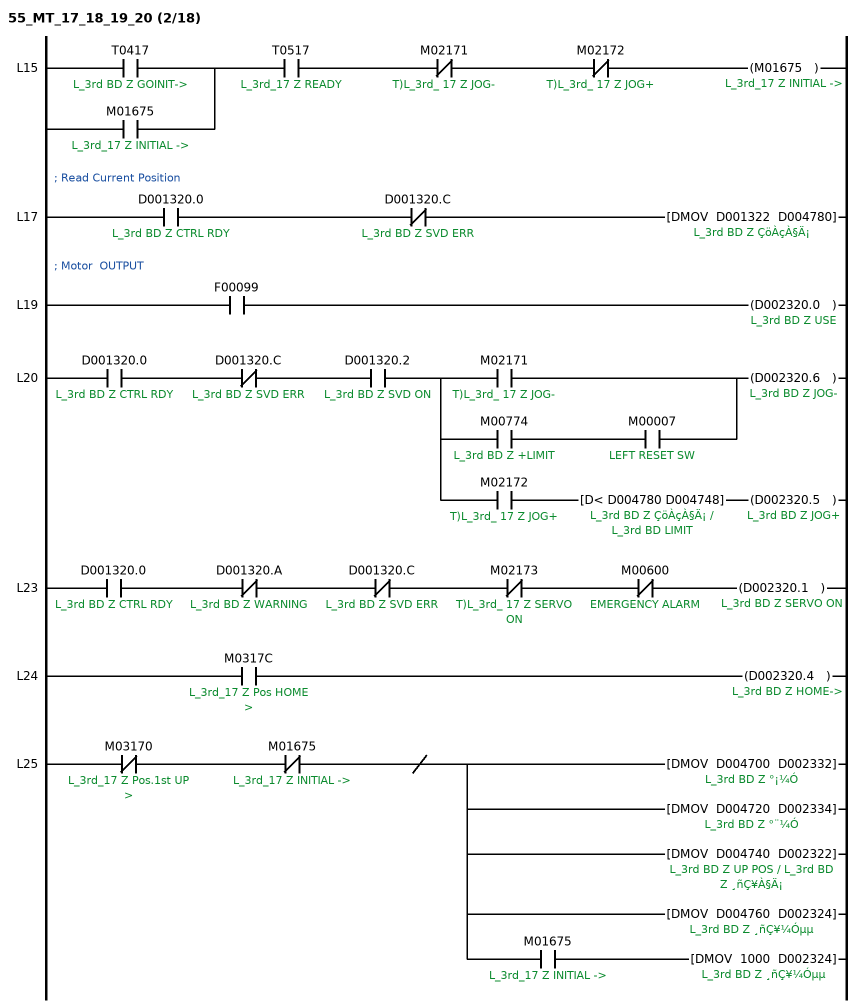
; L15
LOAD      T0417	// L_3rd BD Z GOINIT->
OR        M01675	// L_3rd_17 Z INITIAL ->
AND       T0517	// L_3rd_17 Z READY
AND NOT   M02171	// T)L_3rd_ 17 Z JOG-
AND NOT   M02172	// T)L_3rd_ 17 Z JOG+
OUT       M01675	// L_3rd_17 Z INITIAL ->
; L17
LOAD      D001320.0	// L_3rd BD Z CTRL RDY
AND NOT   D001320.C	// L_3rd BD Z SVD ERR
DMOV      D001322 D004780	// L_3rd BD Z ÇöÀçÀ§Ä¡
// output comment: Read Current Position
//  Motor  OUTPUT
; L19
LOAD      F00099
OUT       D002320.0	// L_3rd BD Z USE
; L20
LOAD      D001320.0	// L_3rd BD Z CTRL RDY
AND NOT   D001320.C	// L_3rd BD Z SVD ERR
AND       D001320.2	// L_3rd BD Z SVD ON
MPUSH
LOAD      M02171	// T)L_3rd_ 17 Z JOG-
LOAD      M00774	// L_3rd BD Z +LIMIT
AND       M00007	// LEFT RESET SW
OR LOAD
AND LOAD
OUT       D002320.6	// L_3rd BD Z JOG-
MPOP
AND       M02172	// T)L_3rd_ 17 Z JOG+
ANDD<     D004780 D004748	// L_3rd BD Z ÇöÀçÀ§Ä¡ / L_3rd BD LIMIT
OUT       D002320.5	// L_3rd BD Z JOG+
; L23
LOAD      D001320.0	// L_3rd BD Z CTRL RDY
AND NOT   D001320.A	// L_3rd BD Z WARNING
AND NOT   D001320.C	// L_3rd BD Z SVD ERR
AND NOT   M02173	// T)L_3rd_ 17 Z SERVO ON
AND NOT   M00600	// EMERGENCY ALARM
OUT       D002320.1	// L_3rd BD Z SERVO ON
; L24
LOAD      M0317C	// L_3rd_17 Z Pos HOME >
OUT       D002320.4	// L_3rd BD Z HOME->
; L25
LOAD NOT  M03170	// L_3rd_17 Z Pos.1st UP >
AND NOT   M01675	// L_3rd_17 Z INITIAL ->
NOT
DMOV      D004700 D002332	// L_3rd BD Z °¡¼Ó
DMOV      D004720 D002334	// L_3rd BD Z °¨¼Ó
DMOV      D004740 D002322	// L_3rd BD Z UP POS / L_3rd BD Z ¸ñÇ¥À§Ä¡
DMOV      D004760 D002324	// L_3rd BD Z ¸ñÇ¥¼Óµµ
AND       M01675	// L_3rd_17 Z INITIAL ->
DMOV      1000 D002324	// L_3rd BD Z ¸ñÇ¥¼Óµµ

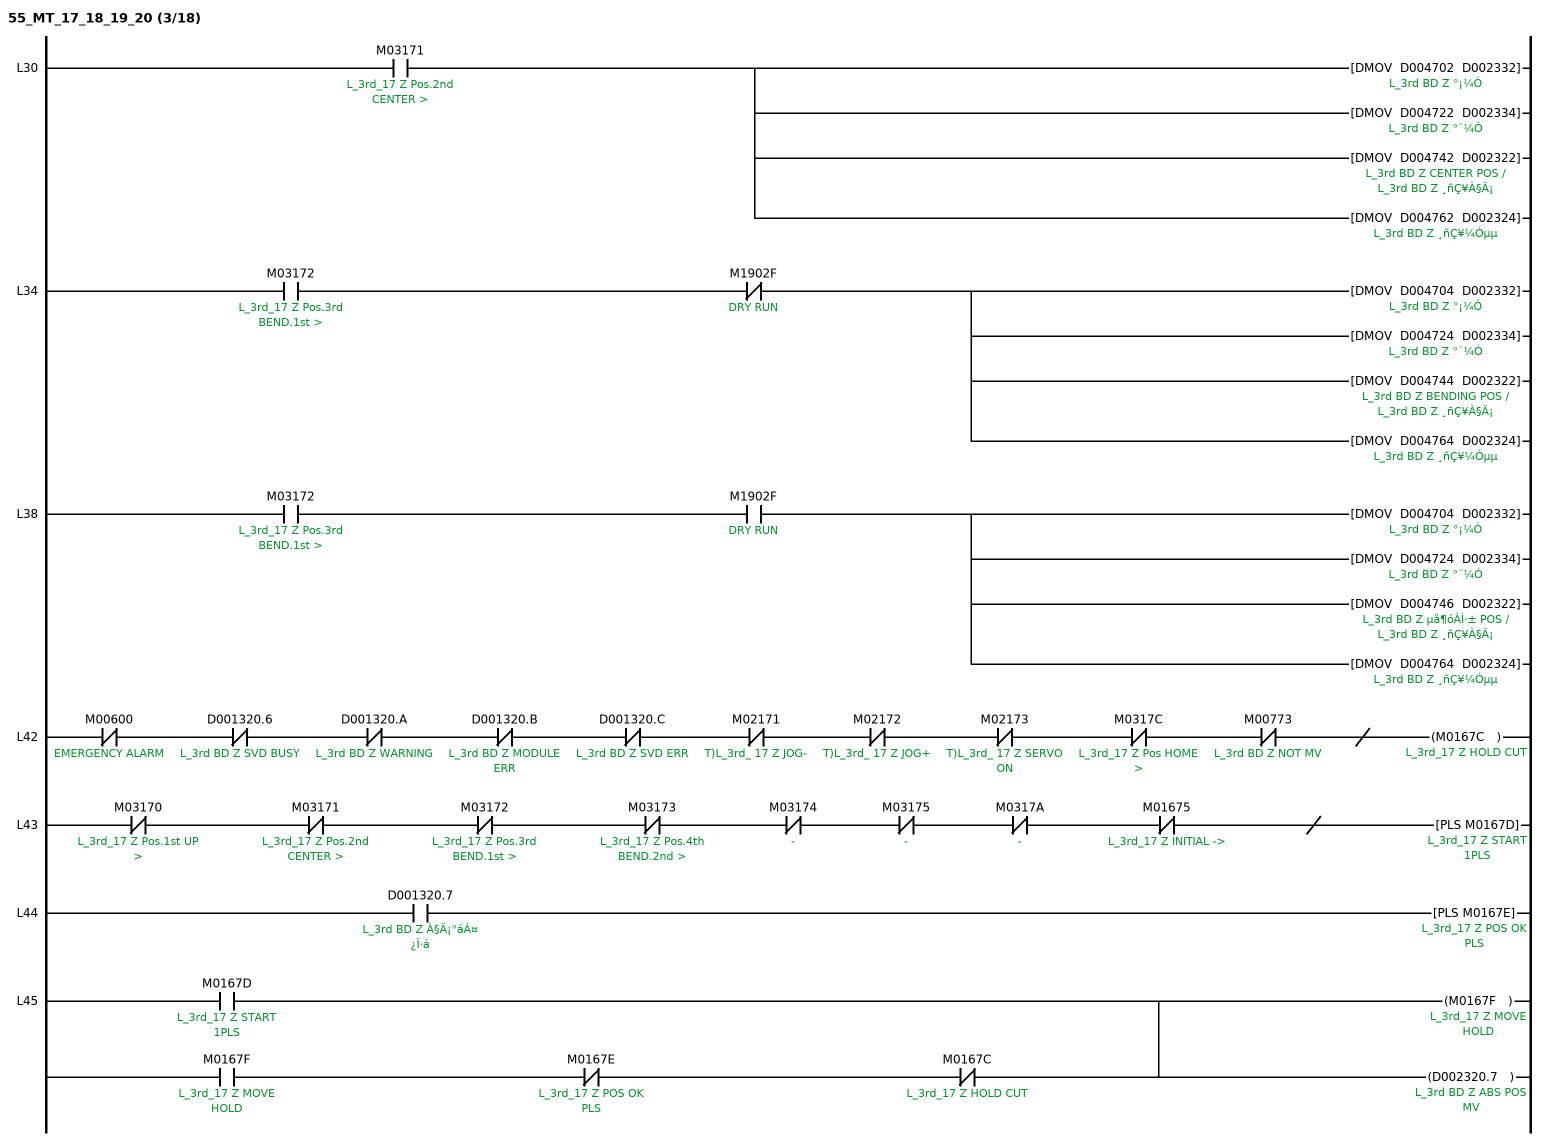
; L30
LOAD      M03171	// L_3rd_17 Z Pos.2nd CENTER >
DMOV      D004702 D002332	// L_3rd BD Z °¡¼Ó
DMOV      D004722 D002334	// L_3rd BD Z °¨¼Ó
DMOV      D004742 D002322	// L_3rd BD Z CENTER POS / L_3rd BD Z ¸ñÇ¥À§Ä¡
DMOV      D004762 D002324	// L_3rd BD Z ¸ñÇ¥¼Óµµ
; L34
LOAD      M03172	// L_3rd_17 Z Pos.3rd BEND.1st >
AND NOT   M1902F	// DRY RUN
DMOV      D004704 D002332	// L_3rd BD Z °¡¼Ó
DMOV      D004724 D002334	// L_3rd BD Z °¨¼Ó
DMOV      D004744 D002322	// L_3rd BD Z BENDING POS / L_3rd BD Z ¸ñÇ¥À§Ä¡
DMOV      D004764 D002324	// L_3rd BD Z ¸ñÇ¥¼Óµµ
; L38
LOAD      M03172	// L_3rd_17 Z Pos.3rd BEND.1st >
AND       M1902F	// DRY RUN
DMOV      D004704 D002332	// L_3rd BD Z °¡¼Ó
DMOV      D004724 D002334	// L_3rd BD Z °¨¼Ó
DMOV      D004746 D002322	// L_3rd BD Z µå¶óÀÌ·± POS / L_3rd BD Z ¸ñÇ¥À§Ä¡
DMOV      D004764 D002324	// L_3rd BD Z ¸ñÇ¥¼Óµµ
; L42
LOAD NOT  M00600	// EMERGENCY ALARM
AND NOT   D001320.6	// L_3rd BD Z SVD BUSY
AND NOT   D001320.A	// L_3rd BD Z WARNING
AND NOT   D001320.B	// L_3rd BD Z MODULE ERR
AND NOT   D001320.C	// L_3rd BD Z SVD ERR
AND NOT   M02171	// T)L_3rd_ 17 Z JOG-
AND NOT   M02172	// T)L_3rd_ 17 Z JOG+
AND NOT   M02173	// T)L_3rd_ 17 Z SERVO ON
AND NOT   M0317C	// L_3rd_17 Z Pos HOME >
AND NOT   M00773	// L_3rd BD Z NOT MV
NOT
OUT       M0167C	// L_3rd_17 Z HOLD CUT
; L43
LOAD NOT  M03170	// L_3rd_17 Z Pos.1st UP >
AND NOT   M03171	// L_3rd_17 Z Pos.2nd CENTER >
AND NOT   M03172	// L_3rd_17 Z Pos.3rd BEND.1st >
AND NOT   M03173	// L_3rd_17 Z Pos.4th BEND.2nd >
AND NOT   M03174	// -
AND NOT   M03175	// -
AND NOT   M0317A	// -
AND NOT   M01675	// L_3rd_17 Z INITIAL ->
NOT
OUTP      M0167D	// L_3rd_17 Z START 1PLS
; L44
LOAD      D001320.7	// L_3rd BD Z À§Ä¡°áÁ¤ ¿Ï·á
OUTP      M0167E	// L_3rd_17 Z POS OK PLS
; L45
LOAD      M0167D	// L_3rd_17 Z START 1PLS
LOAD      M0167F	// L_3rd_17 Z MOVE HOLD
AND NOT   M0167E	// L_3rd_17 Z POS OK PLS
AND NOT   M0167C	// L_3rd_17 Z HOLD CUT
OR LOAD
OUT       M0167F	// L_3rd_17 Z MOVE HOLD
OUT       D002320.7	// L_3rd BD Z ABS POS MV

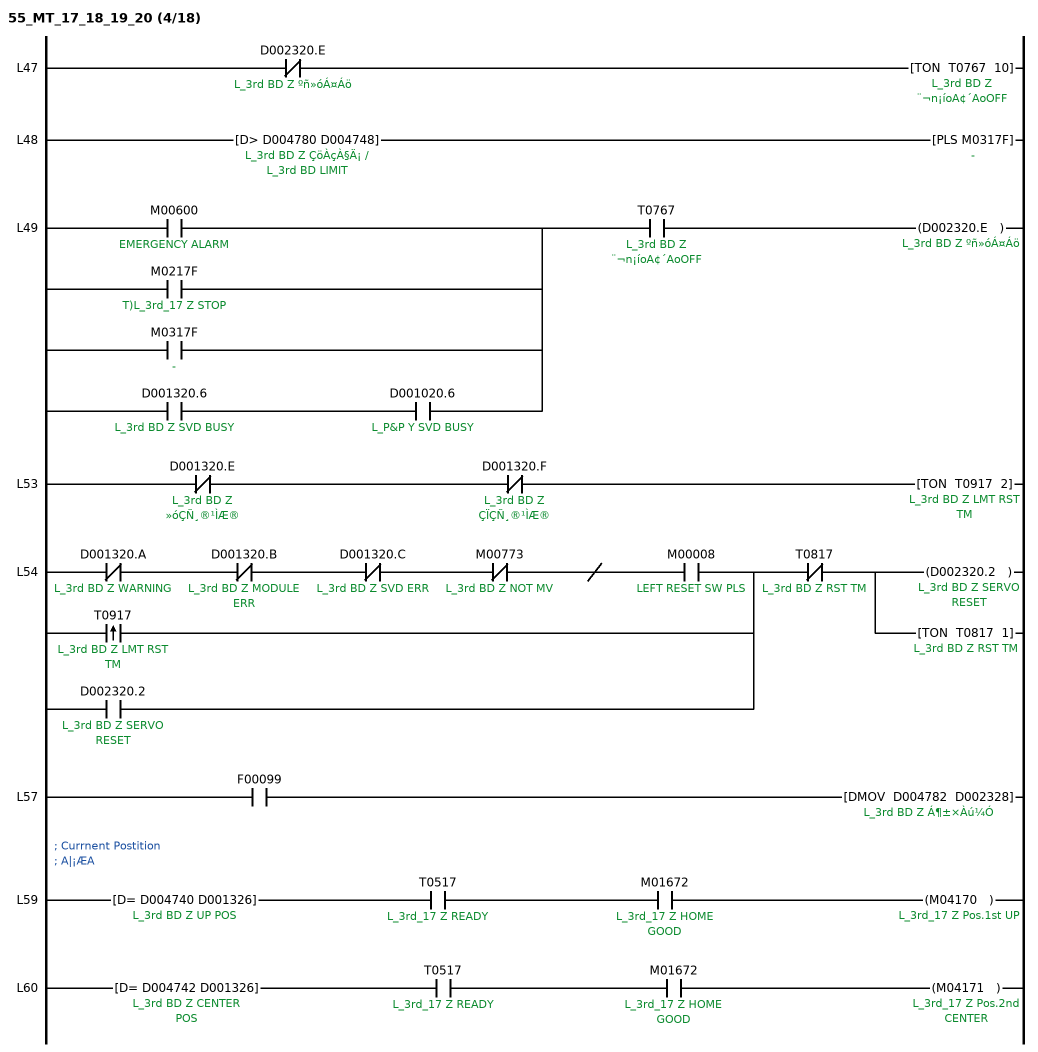
; L47
LOAD NOT  D002320.E	// L_3rd BD Z ºñ»óÁ¤Áö
TON       T0767 10	// L_3rd BD Z ¨¬n¡íoA¢´AoOFF
; L48
LOADD>    D004780 D004748	// L_3rd BD Z ÇöÀçÀ§Ä¡ / L_3rd BD LIMIT
OUTP      M0317F	// -
; L49
LOAD      M00600	// EMERGENCY ALARM
OR        M0217F	// T)L_3rd_17 Z STOP
OR        M0317F	// -
LOAD      D001320.6	// L_3rd BD Z SVD BUSY
AND       D001020.6	// L_P&P Y SVD BUSY
OR LOAD
AND       T0767	// L_3rd BD Z ¨¬n¡íoA¢´AoOFF
OUT       D002320.E	// L_3rd BD Z ºñ»óÁ¤Áö
; L53
LOAD NOT  D001320.E	// L_3rd BD Z »óÇÑ¸®¹ÌÆ®
AND NOT   D001320.F	// L_3rd BD Z ÇÏÇÑ¸®¹ÌÆ®
TON       T0917 2	// L_3rd BD Z LMT RST TM
; L54
LOAD NOT  D001320.A	// L_3rd BD Z WARNING
AND NOT   D001320.B	// L_3rd BD Z MODULE ERR
AND NOT   D001320.C	// L_3rd BD Z SVD ERR
AND NOT   M00773	// L_3rd BD Z NOT MV
NOT
AND       M00008	// LEFT RESET SW PLS
ORP       T0917	// L_3rd BD Z LMT RST TM
OR        D002320.2	// L_3rd BD Z SERVO RESET
AND NOT   T0817	// L_3rd BD Z RST TM
OUT       D002320.2	// L_3rd BD Z SERVO RESET
TON       T0817 1	// L_3rd BD Z RST TM
; L57
LOAD      F00099
DMOV      D004782 D002328	// L_3rd BD Z Á¶±×Àú¼Ó
// Currnent Postition
; L59
LOADD=    D004740 D001326	// L_3rd BD Z UP POS
AND       T0517	// L_3rd_17 Z READY
AND       M01672	// L_3rd_17 Z HOME GOOD
OUT       M04170	// L_3rd_17 Z Pos.1st UP
// output comment: A|¡ÆA
; L60
LOADD=    D004742 D001326	// L_3rd BD Z CENTER POS
AND       T0517	// L_3rd_17 Z READY
AND       M01672	// L_3rd_17 Z HOME GOOD
OUT       M04171	// L_3rd_17 Z Pos.2nd CENTER

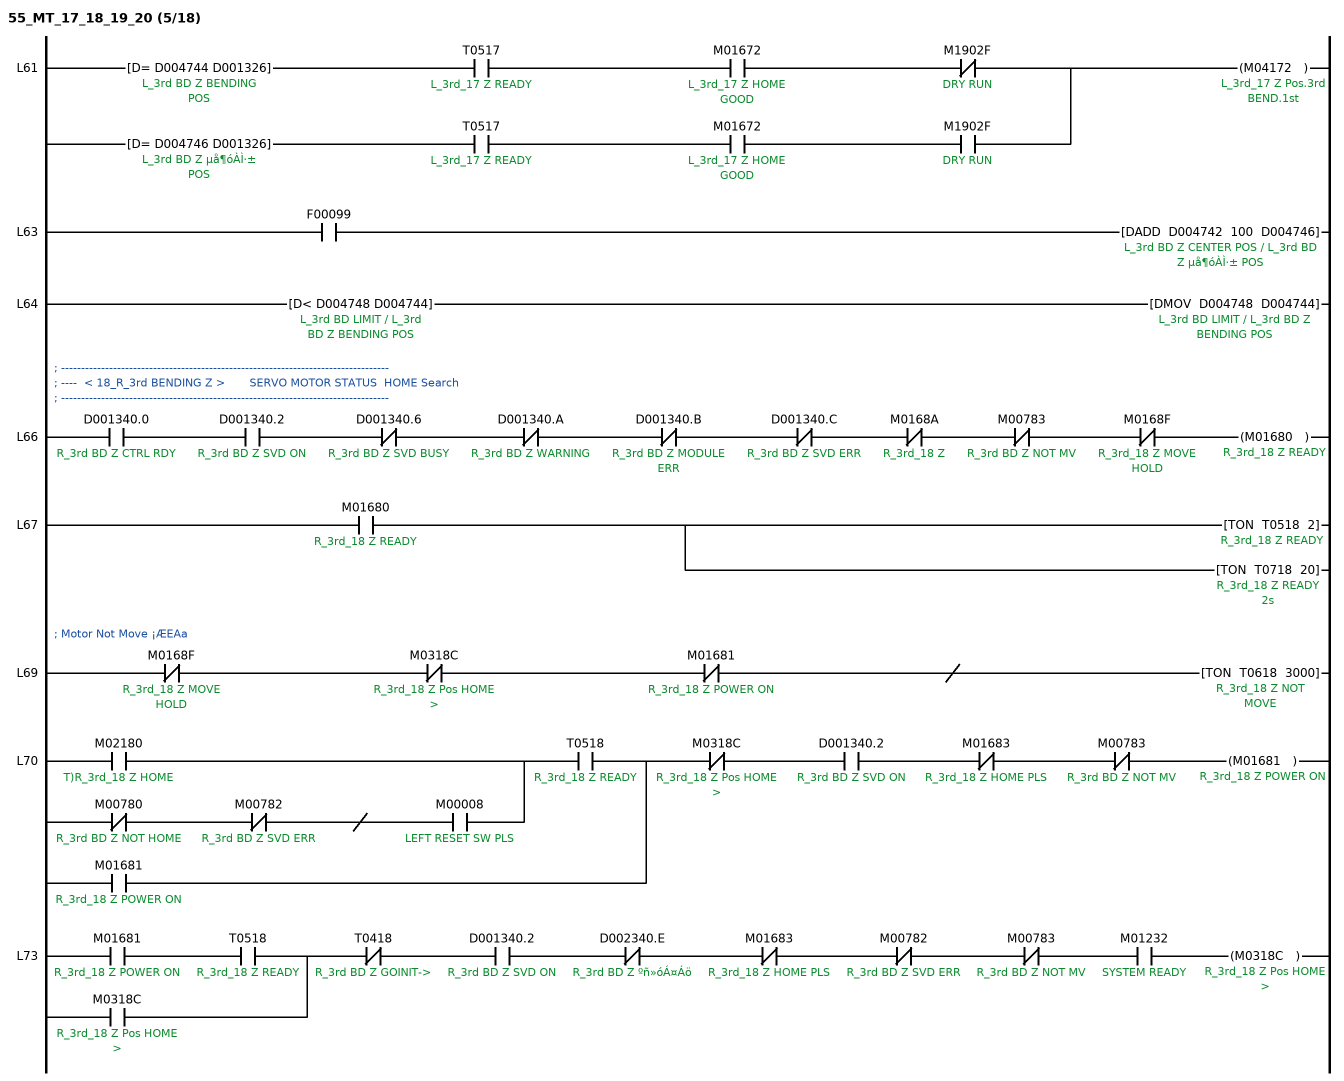
; L61
LOADD=    D004744 D001326	// L_3rd BD Z BENDING POS
AND       T0517	// L_3rd_17 Z READY
AND       M01672	// L_3rd_17 Z HOME GOOD
AND NOT   M1902F	// DRY RUN
LOADD=    D004746 D001326	// L_3rd BD Z µå¶óÀÌ·± POS
AND       T0517	// L_3rd_17 Z READY
AND       M01672	// L_3rd_17 Z HOME GOOD
AND       M1902F	// DRY RUN
OR LOAD
OUT       M04172	// L_3rd_17 Z Pos.3rd BEND.1st
; L63
LOAD      F00099
DADD      D004742 100 D004746	// L_3rd BD Z CENTER POS / L_3rd BD Z µå¶óÀÌ·± POS
; L64
LOADD<    D004748 D004744	// L_3rd BD LIMIT / L_3rd BD Z BENDING POS
DMOV      D004748 D004744	// L_3rd BD LIMIT / L_3rd BD Z BENDING POS
// ----------------------------------------------------------------------------------
// 
// ----  < 18_R_3rd BENDING Z >       SERVO MOTOR STATUS  HOME Search
// 
// ----------------------------------------------------------------------------------
; L66
LOAD      D001340.0	// R_3rd BD Z CTRL RDY
AND       D001340.2	// R_3rd BD Z SVD ON
AND NOT   D001340.6	// R_3rd BD Z SVD BUSY
AND NOT   D001340.A	// R_3rd BD Z WARNING
AND NOT   D001340.B	// R_3rd BD Z MODULE ERR
AND NOT   D001340.C	// R_3rd BD Z SVD ERR
AND NOT   M0168A	// R_3rd_18 Z
AND NOT   M00783	// R_3rd BD Z NOT MV
AND NOT   M0168F	// R_3rd_18 Z MOVE HOLD
OUT       M01680	// R_3rd_18 Z READY
; L67
LOAD      M01680	// R_3rd_18 Z READY
TON       T0518 2	// R_3rd_18 Z READY
TON       T0718 20	// R_3rd_18 Z READY 2s
; L69
LOAD NOT  M0168F	// R_3rd_18 Z MOVE HOLD
AND NOT   M0318C	// R_3rd_18 Z Pos HOME >
AND NOT   M01681	// R_3rd_18 Z POWER ON
NOT
TON       T0618 3000	// R_3rd_18 Z NOT MOVE
// output comment: Motor Not Move ¡ÆEAa
; L70
LOAD      M02180	// T)R_3rd_18 Z HOME
LOAD NOT  M00780	// R_3rd BD Z NOT HOME
AND NOT   M00782	// R_3rd BD Z SVD ERR
NOT
AND       M00008	// LEFT RESET SW PLS
OR LOAD
AND       T0518	// R_3rd_18 Z READY
OR        M01681	// R_3rd_18 Z POWER ON
AND NOT   M0318C	// R_3rd_18 Z Pos HOME >
AND       D001340.2	// R_3rd BD Z SVD ON
AND NOT   M01683	// R_3rd_18 Z HOME PLS
AND NOT   M00783	// R_3rd BD Z NOT MV
OUT       M01681	// R_3rd_18 Z POWER ON
; L73
LOAD      M01681	// R_3rd_18 Z POWER ON
AND       T0518	// R_3rd_18 Z READY
OR        M0318C	// R_3rd_18 Z Pos HOME >
AND NOT   T0418	// R_3rd BD Z GOINIT->
AND       D001340.2	// R_3rd BD Z SVD ON
AND NOT   D002340.E	// R_3rd BD Z ºñ»óÁ¤Áö
AND NOT   M01683	// R_3rd_18 Z HOME PLS
AND NOT   M00782	// R_3rd BD Z SVD ERR
AND NOT   M00783	// R_3rd BD Z NOT MV
AND       M01232	// SYSTEM READY
OUT       M0318C	// R_3rd_18 Z Pos HOME >

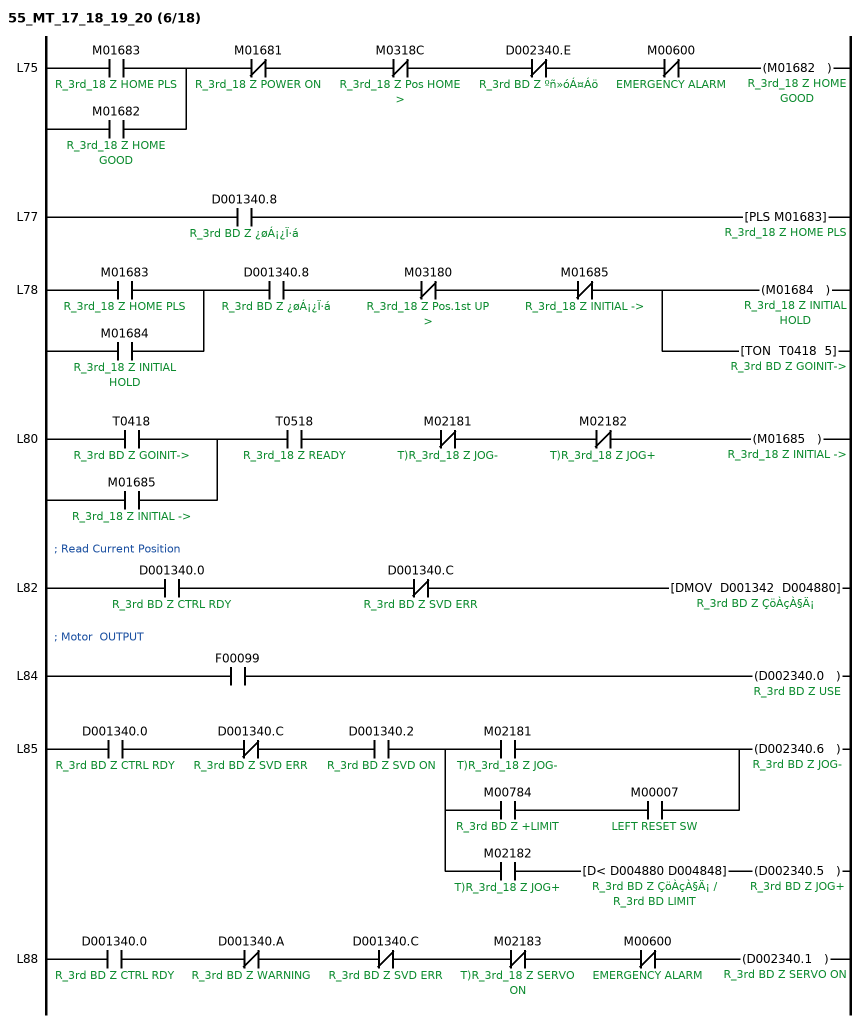
; L75
LOAD      M01683	// R_3rd_18 Z HOME PLS
OR        M01682	// R_3rd_18 Z HOME GOOD
AND NOT   M01681	// R_3rd_18 Z POWER ON
AND NOT   M0318C	// R_3rd_18 Z Pos HOME >
AND NOT   D002340.E	// R_3rd BD Z ºñ»óÁ¤Áö
AND NOT   M00600	// EMERGENCY ALARM
OUT       M01682	// R_3rd_18 Z HOME GOOD
; L77
LOAD      D001340.8	// R_3rd BD Z ¿øÁ¡¿Ï·á
OUTP      M01683	// R_3rd_18 Z HOME PLS
; L78
LOAD      M01683	// R_3rd_18 Z HOME PLS
OR        M01684	// R_3rd_18 Z INITIAL HOLD
AND       D001340.8	// R_3rd BD Z ¿øÁ¡¿Ï·á
AND NOT   M03180	// R_3rd_18 Z Pos.1st UP >
AND NOT   M01685	// R_3rd_18 Z INITIAL ->
OUT       M01684	// R_3rd_18 Z INITIAL HOLD
TON       T0418 5	// R_3rd BD Z GOINIT->
; L80
LOAD      T0418	// R_3rd BD Z GOINIT->
OR        M01685	// R_3rd_18 Z INITIAL ->
AND       T0518	// R_3rd_18 Z READY
AND NOT   M02181	// T)R_3rd_18 Z JOG-
AND NOT   M02182	// T)R_3rd_18 Z JOG+
OUT       M01685	// R_3rd_18 Z INITIAL ->
; L82
LOAD      D001340.0	// R_3rd BD Z CTRL RDY
AND NOT   D001340.C	// R_3rd BD Z SVD ERR
DMOV      D001342 D004880	// R_3rd BD Z ÇöÀçÀ§Ä¡
// output comment: Read Current Position
//  Motor  OUTPUT
; L84
LOAD      F00099
OUT       D002340.0	// R_3rd BD Z USE
; L85
LOAD      D001340.0	// R_3rd BD Z CTRL RDY
AND NOT   D001340.C	// R_3rd BD Z SVD ERR
AND       D001340.2	// R_3rd BD Z SVD ON
MPUSH
LOAD      M02181	// T)R_3rd_18 Z JOG-
LOAD      M00784	// R_3rd BD Z +LIMIT
AND       M00007	// LEFT RESET SW
OR LOAD
AND LOAD
OUT       D002340.6	// R_3rd BD Z JOG-
MPOP
AND       M02182	// T)R_3rd_18 Z JOG+
ANDD<     D004880 D004848	// R_3rd BD Z ÇöÀçÀ§Ä¡ / R_3rd BD LIMIT
OUT       D002340.5	// R_3rd BD Z JOG+
; L88
LOAD      D001340.0	// R_3rd BD Z CTRL RDY
AND NOT   D001340.A	// R_3rd BD Z WARNING
AND NOT   D001340.C	// R_3rd BD Z SVD ERR
AND NOT   M02183	// T)R_3rd_18 Z SERVO ON
AND NOT   M00600	// EMERGENCY ALARM
OUT       D002340.1	// R_3rd BD Z SERVO ON

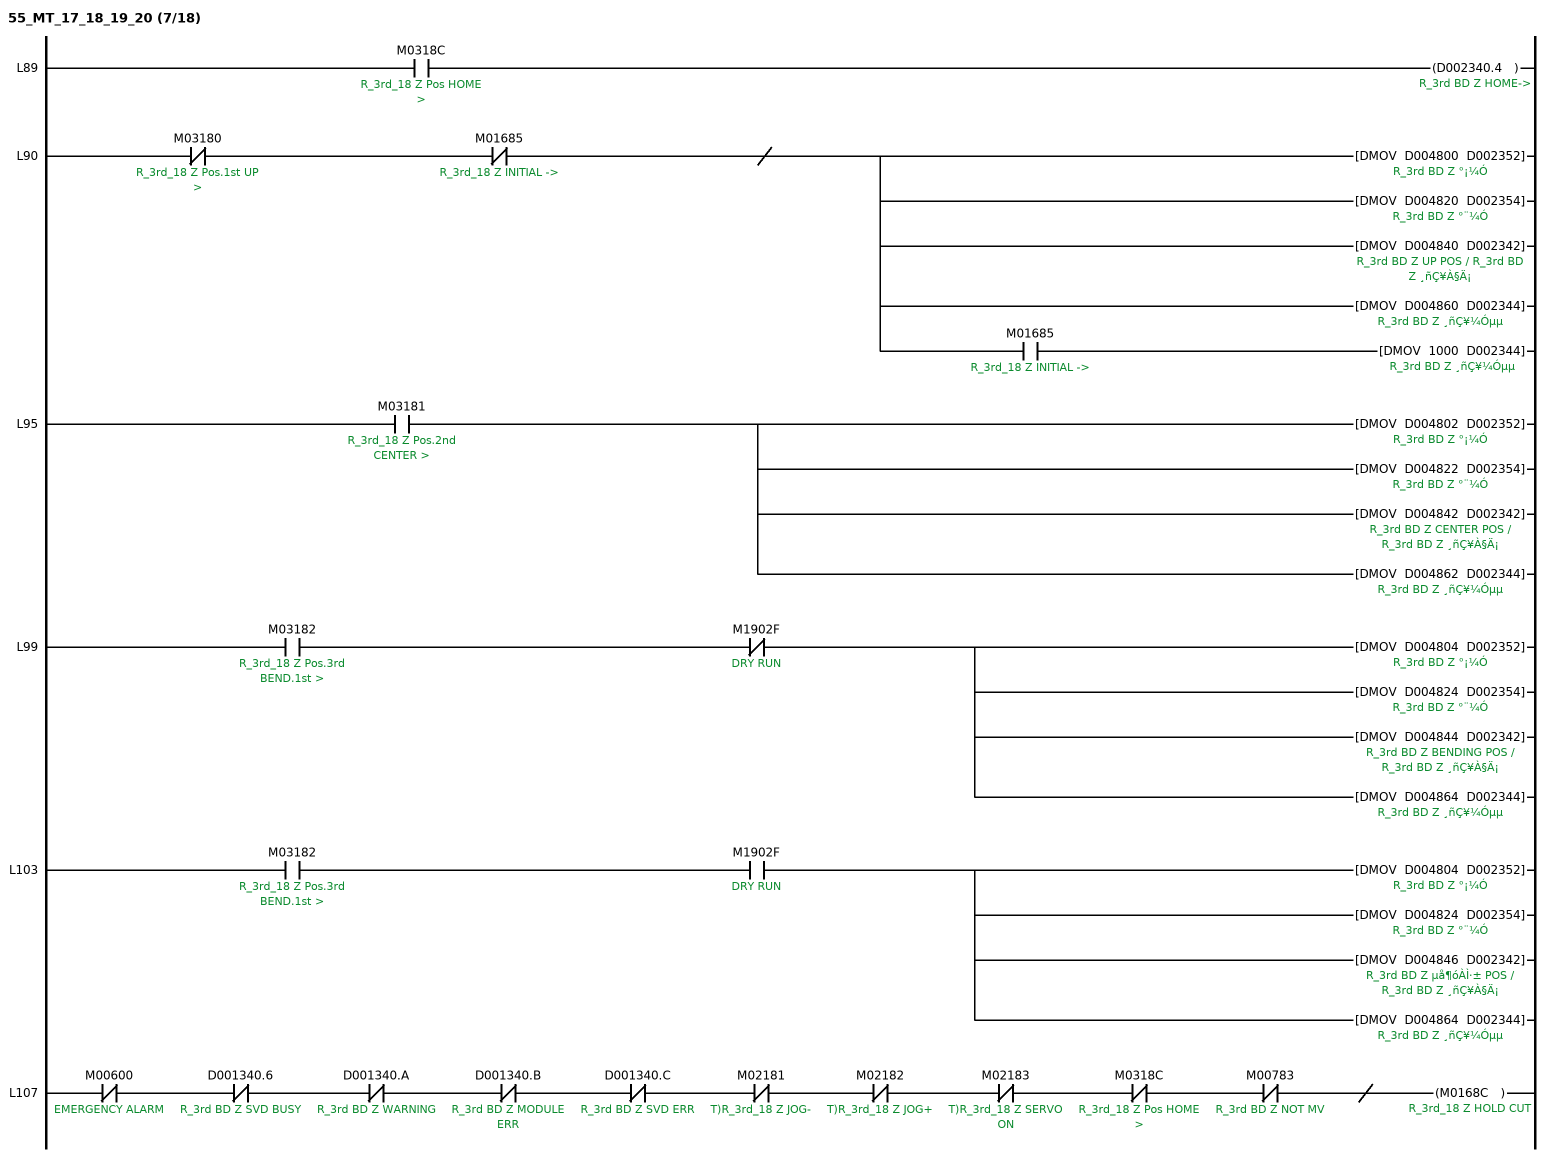
; L89
LOAD      M0318C	// R_3rd_18 Z Pos HOME >
OUT       D002340.4	// R_3rd BD Z HOME->
; L90
LOAD NOT  M03180	// R_3rd_18 Z Pos.1st UP >
AND NOT   M01685	// R_3rd_18 Z INITIAL ->
NOT
DMOV      D004800 D002352	// R_3rd BD Z °¡¼Ó
DMOV      D004820 D002354	// R_3rd BD Z °¨¼Ó
DMOV      D004840 D002342	// R_3rd BD Z UP POS / R_3rd BD Z ¸ñÇ¥À§Ä¡
DMOV      D004860 D002344	// R_3rd BD Z ¸ñÇ¥¼Óµµ
AND       M01685	// R_3rd_18 Z INITIAL ->
DMOV      1000 D002344	// R_3rd BD Z ¸ñÇ¥¼Óµµ
; L95
LOAD      M03181	// R_3rd_18 Z Pos.2nd CENTER >
DMOV      D004802 D002352	// R_3rd BD Z °¡¼Ó
DMOV      D004822 D002354	// R_3rd BD Z °¨¼Ó
DMOV      D004842 D002342	// R_3rd BD Z CENTER POS / R_3rd BD Z ¸ñÇ¥À§Ä¡
DMOV      D004862 D002344	// R_3rd BD Z ¸ñÇ¥¼Óµµ
; L99
LOAD      M03182	// R_3rd_18 Z Pos.3rd BEND.1st >
AND NOT   M1902F	// DRY RUN
DMOV      D004804 D002352	// R_3rd BD Z °¡¼Ó
DMOV      D004824 D002354	// R_3rd BD Z °¨¼Ó
DMOV      D004844 D002342	// R_3rd BD Z BENDING POS / R_3rd BD Z ¸ñÇ¥À§Ä¡
DMOV      D004864 D002344	// R_3rd BD Z ¸ñÇ¥¼Óµµ
; L103
LOAD      M03182	// R_3rd_18 Z Pos.3rd BEND.1st >
AND       M1902F	// DRY RUN
DMOV      D004804 D002352	// R_3rd BD Z °¡¼Ó
DMOV      D004824 D002354	// R_3rd BD Z °¨¼Ó
DMOV      D004846 D002342	// R_3rd BD Z µå¶óÀÌ·± POS / R_3rd BD Z ¸ñÇ¥À§Ä¡
DMOV      D004864 D002344	// R_3rd BD Z ¸ñÇ¥¼Óµµ
; L107
LOAD NOT  M00600	// EMERGENCY ALARM
AND NOT   D001340.6	// R_3rd BD Z SVD BUSY
AND NOT   D001340.A	// R_3rd BD Z WARNING
AND NOT   D001340.B	// R_3rd BD Z MODULE ERR
AND NOT   D001340.C	// R_3rd BD Z SVD ERR
AND NOT   M02181	// T)R_3rd_18 Z JOG-
AND NOT   M02182	// T)R_3rd_18 Z JOG+
AND NOT   M02183	// T)R_3rd_18 Z SERVO ON
AND NOT   M0318C	// R_3rd_18 Z Pos HOME >
AND NOT   M00783	// R_3rd BD Z NOT MV
NOT
OUT       M0168C	// R_3rd_18 Z HOLD CUT

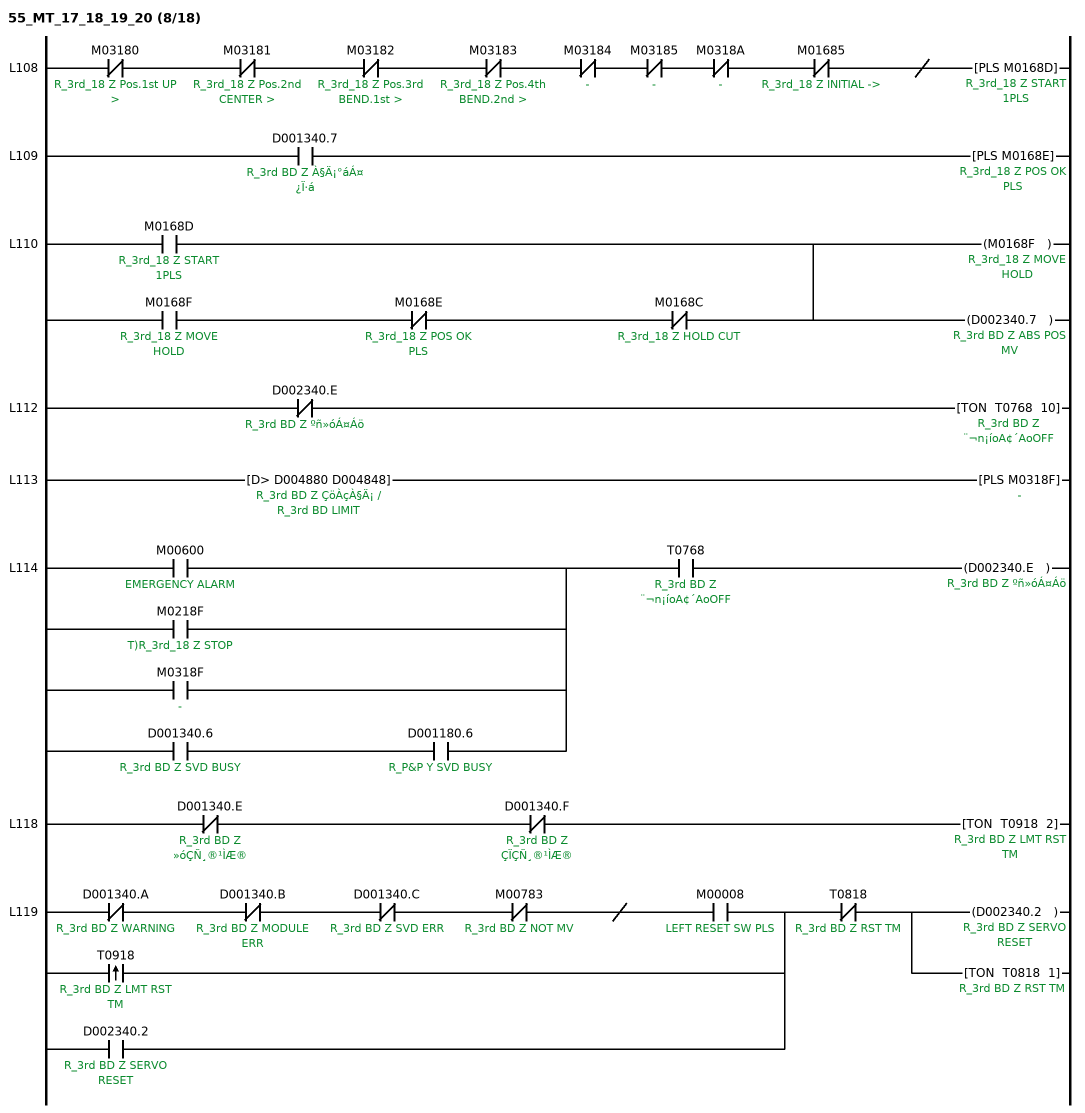
; L108
LOAD NOT  M03180	// R_3rd_18 Z Pos.1st UP >
AND NOT   M03181	// R_3rd_18 Z Pos.2nd CENTER >
AND NOT   M03182	// R_3rd_18 Z Pos.3rd BEND.1st >
AND NOT   M03183	// R_3rd_18 Z Pos.4th BEND.2nd >
AND NOT   M03184	// -
AND NOT   M03185	// -
AND NOT   M0318A	// -
AND NOT   M01685	// R_3rd_18 Z INITIAL ->
NOT
OUTP      M0168D	// R_3rd_18 Z START 1PLS
; L109
LOAD      D001340.7	// R_3rd BD Z À§Ä¡°áÁ¤ ¿Ï·á
OUTP      M0168E	// R_3rd_18 Z POS OK PLS
; L110
LOAD      M0168D	// R_3rd_18 Z START 1PLS
LOAD      M0168F	// R_3rd_18 Z MOVE HOLD
AND NOT   M0168E	// R_3rd_18 Z POS OK PLS
AND NOT   M0168C	// R_3rd_18 Z HOLD CUT
OR LOAD
OUT       M0168F	// R_3rd_18 Z MOVE HOLD
OUT       D002340.7	// R_3rd BD Z ABS POS MV
; L112
LOAD NOT  D002340.E	// R_3rd BD Z ºñ»óÁ¤Áö
TON       T0768 10	// R_3rd BD Z ¨¬n¡íoA¢´AoOFF
; L113
LOADD>    D004880 D004848	// R_3rd BD Z ÇöÀçÀ§Ä¡ / R_3rd BD LIMIT
OUTP      M0318F	// -
; L114
LOAD      M00600	// EMERGENCY ALARM
OR        M0218F	// T)R_3rd_18 Z STOP
OR        M0318F	// -
LOAD      D001340.6	// R_3rd BD Z SVD BUSY
AND       D001180.6	// R_P&P Y SVD BUSY
OR LOAD
AND       T0768	// R_3rd BD Z ¨¬n¡íoA¢´AoOFF
OUT       D002340.E	// R_3rd BD Z ºñ»óÁ¤Áö
; L118
LOAD NOT  D001340.E	// R_3rd BD Z »óÇÑ¸®¹ÌÆ®
AND NOT   D001340.F	// R_3rd BD Z ÇÏÇÑ¸®¹ÌÆ®
TON       T0918 2	// R_3rd BD Z LMT RST TM
; L119
LOAD NOT  D001340.A	// R_3rd BD Z WARNING
AND NOT   D001340.B	// R_3rd BD Z MODULE ERR
AND NOT   D001340.C	// R_3rd BD Z SVD ERR
AND NOT   M00783	// R_3rd BD Z NOT MV
NOT
AND       M00008	// LEFT RESET SW PLS
ORP       T0918	// R_3rd BD Z LMT RST TM
OR        D002340.2	// R_3rd BD Z SERVO RESET
AND NOT   T0818	// R_3rd BD Z RST TM
OUT       D002340.2	// R_3rd BD Z SERVO RESET
TON       T0818 1	// R_3rd BD Z RST TM

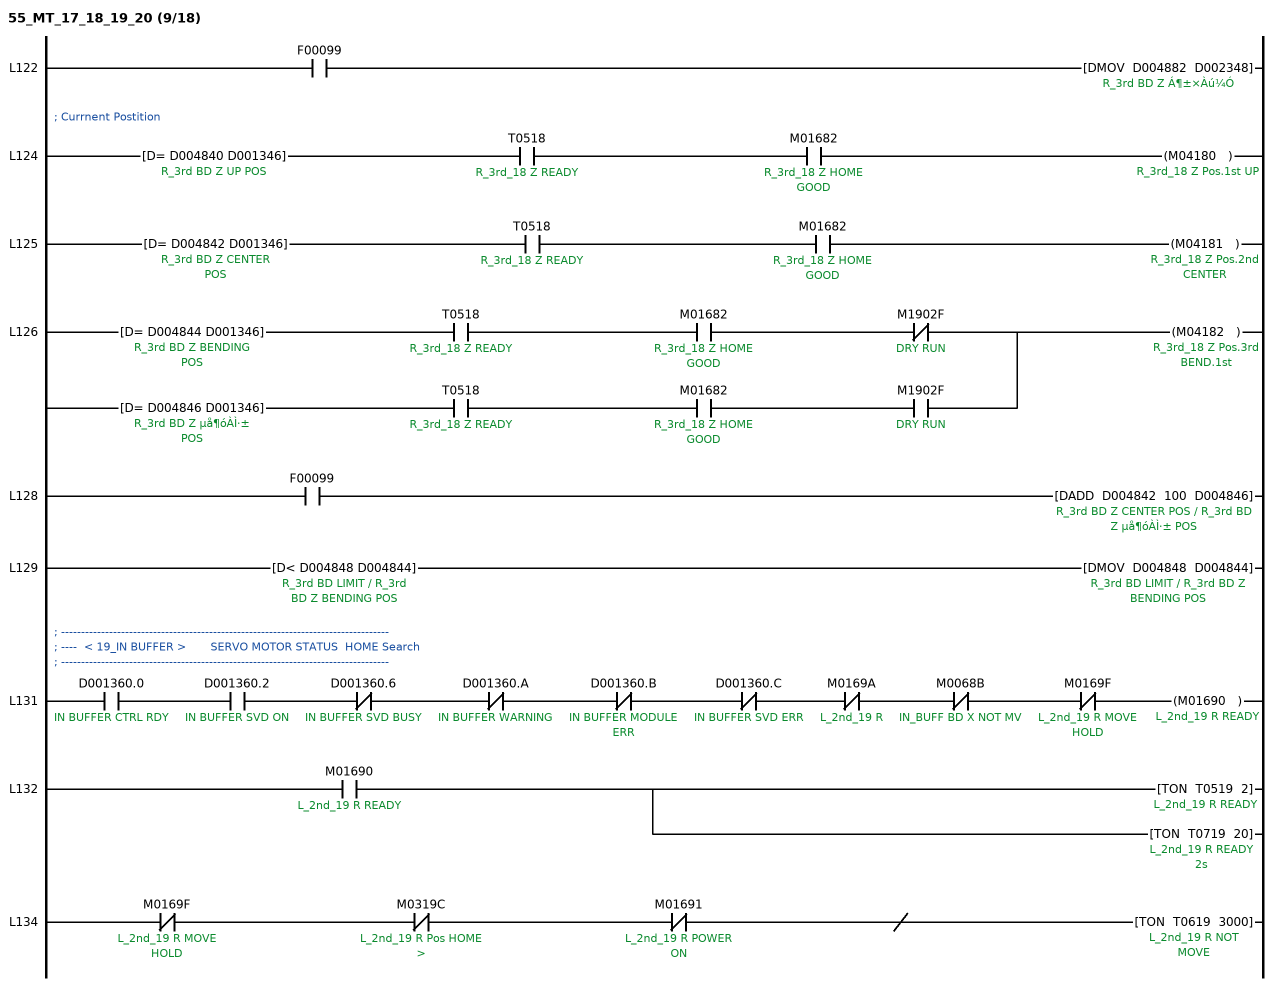
; L122
LOAD      F00099
DMOV      D004882 D002348	// R_3rd BD Z Á¶±×Àú¼Ó
// Currnent Postition
; L124
LOADD=    D004840 D001346	// R_3rd BD Z UP POS
AND       T0518	// R_3rd_18 Z READY
AND       M01682	// R_3rd_18 Z HOME GOOD
OUT       M04180	// R_3rd_18 Z Pos.1st UP
; L125
LOADD=    D004842 D001346	// R_3rd BD Z CENTER POS
AND       T0518	// R_3rd_18 Z READY
AND       M01682	// R_3rd_18 Z HOME GOOD
OUT       M04181	// R_3rd_18 Z Pos.2nd CENTER
; L126
LOADD=    D004844 D001346	// R_3rd BD Z BENDING POS
AND       T0518	// R_3rd_18 Z READY
AND       M01682	// R_3rd_18 Z HOME GOOD
AND NOT   M1902F	// DRY RUN
LOADD=    D004846 D001346	// R_3rd BD Z µå¶óÀÌ·± POS
AND       T0518	// R_3rd_18 Z READY
AND       M01682	// R_3rd_18 Z HOME GOOD
AND       M1902F	// DRY RUN
OR LOAD
OUT       M04182	// R_3rd_18 Z Pos.3rd BEND.1st
; L128
LOAD      F00099
DADD      D004842 100 D004846	// R_3rd BD Z CENTER POS / R_3rd BD Z µå¶óÀÌ·± POS
; L129
LOADD<    D004848 D004844	// R_3rd BD LIMIT / R_3rd BD Z BENDING POS
DMOV      D004848 D004844	// R_3rd BD LIMIT / R_3rd BD Z BENDING POS
// ----------------------------------------------------------------------------------
// 
// ----  < 19_IN BUFFER >       SERVO MOTOR STATUS  HOME Search
// 
// ----------------------------------------------------------------------------------
; L131
LOAD      D001360.0	// IN BUFFER CTRL RDY
AND       D001360.2	// IN BUFFER SVD ON
AND NOT   D001360.6	// IN BUFFER SVD BUSY
AND NOT   D001360.A	// IN BUFFER WARNING
AND NOT   D001360.B	// IN BUFFER MODULE ERR
AND NOT   D001360.C	// IN BUFFER SVD ERR
AND NOT   M0169A	// L_2nd_19 R
AND NOT   M0068B	// IN_BUFF BD X NOT MV
AND NOT   M0169F	// L_2nd_19 R MOVE HOLD
OUT       M01690	// L_2nd_19 R READY
; L132
LOAD      M01690	// L_2nd_19 R READY
TON       T0519 2	// L_2nd_19 R READY
TON       T0719 20	// L_2nd_19 R READY 2s
; L134
LOAD NOT  M0169F	// L_2nd_19 R MOVE HOLD
AND NOT   M0319C	// L_2nd_19 R Pos HOME >
AND NOT   M01691	// L_2nd_19 R POWER ON
NOT
TON       T0619 3000	// L_2nd_19 R NOT MOVE

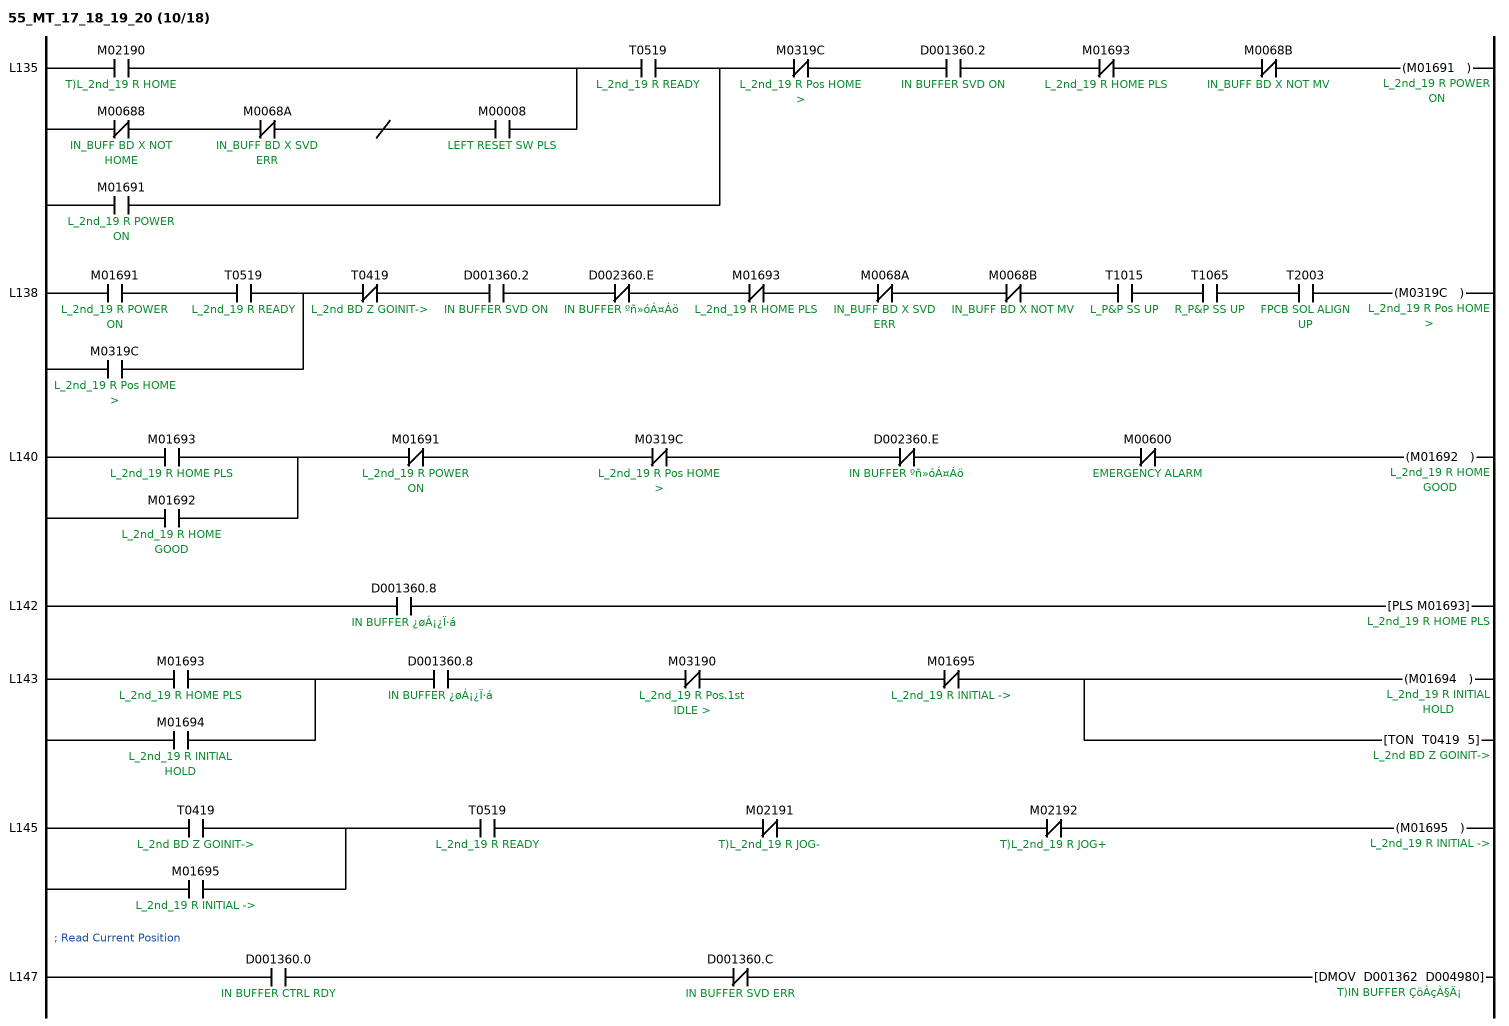
; L135
LOAD      M02190	// T)L_2nd_19 R HOME
LOAD NOT  M00688	// IN_BUFF BD X NOT HOME
AND NOT   M0068A	// IN_BUFF BD X SVD ERR
NOT
AND       M00008	// LEFT RESET SW PLS
OR LOAD
AND       T0519	// L_2nd_19 R READY
OR        M01691	// L_2nd_19 R POWER ON
AND NOT   M0319C	// L_2nd_19 R Pos HOME >
AND       D001360.2	// IN BUFFER SVD ON
AND NOT   M01693	// L_2nd_19 R HOME PLS
AND NOT   M0068B	// IN_BUFF BD X NOT MV
OUT       M01691	// L_2nd_19 R POWER ON
; L138
LOAD      M01691	// L_2nd_19 R POWER ON
AND       T0519	// L_2nd_19 R READY
OR        M0319C	// L_2nd_19 R Pos HOME >
AND NOT   T0419	// L_2nd BD Z GOINIT->
AND       D001360.2	// IN BUFFER SVD ON
AND NOT   D002360.E	// IN BUFFER ºñ»óÁ¤Áö
AND NOT   M01693	// L_2nd_19 R HOME PLS
AND NOT   M0068A	// IN_BUFF BD X SVD ERR
AND NOT   M0068B	// IN_BUFF BD X NOT MV
AND       T1015	// L_P&P SS UP
AND       T1065	// R_P&P SS UP
AND       T2003	// FPCB SOL ALIGN         UP
OUT       M0319C	// L_2nd_19 R Pos HOME >
; L140
LOAD      M01693	// L_2nd_19 R HOME PLS
OR        M01692	// L_2nd_19 R HOME GOOD
AND NOT   M01691	// L_2nd_19 R POWER ON
AND NOT   M0319C	// L_2nd_19 R Pos HOME >
AND NOT   D002360.E	// IN BUFFER ºñ»óÁ¤Áö
AND NOT   M00600	// EMERGENCY ALARM
OUT       M01692	// L_2nd_19 R HOME GOOD
; L142
LOAD      D001360.8	// IN BUFFER ¿øÁ¡¿Ï·á
OUTP      M01693	// L_2nd_19 R HOME PLS
; L143
LOAD      M01693	// L_2nd_19 R HOME PLS
OR        M01694	// L_2nd_19 R INITIAL HOLD
AND       D001360.8	// IN BUFFER ¿øÁ¡¿Ï·á
AND NOT   M03190	// L_2nd_19 R Pos.1st IDLE >
AND NOT   M01695	// L_2nd_19 R INITIAL ->
OUT       M01694	// L_2nd_19 R INITIAL HOLD
TON       T0419 5	// L_2nd BD Z GOINIT->
; L145
LOAD      T0419	// L_2nd BD Z GOINIT->
OR        M01695	// L_2nd_19 R INITIAL ->
AND       T0519	// L_2nd_19 R READY
AND NOT   M02191	// T)L_2nd_19 R JOG-
AND NOT   M02192	// T)L_2nd_19 R JOG+
OUT       M01695	// L_2nd_19 R INITIAL ->
; L147
LOAD      D001360.0	// IN BUFFER CTRL RDY
AND NOT   D001360.C	// IN BUFFER SVD ERR
DMOV      D001362 D004980	// T)IN BUFFER ÇöÀçÀ§Ä¡
// output comment: Read Current Position

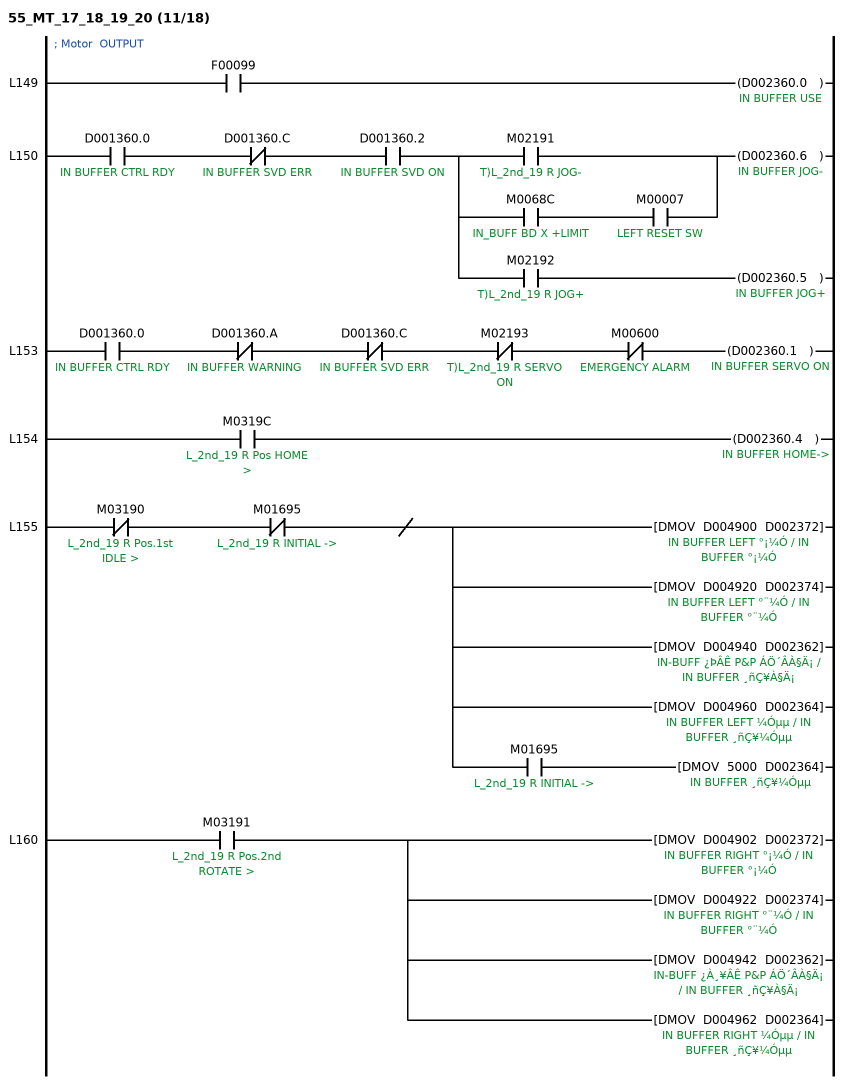
//  Motor  OUTPUT
; L149
LOAD      F00099
OUT       D002360.0	// IN BUFFER USE
; L150
LOAD      D001360.0	// IN BUFFER CTRL RDY
AND NOT   D001360.C	// IN BUFFER SVD ERR
AND       D001360.2	// IN BUFFER SVD ON
MPUSH
LOAD      M02191	// T)L_2nd_19 R JOG-
LOAD      M0068C	// IN_BUFF BD X +LIMIT
AND       M00007	// LEFT RESET SW
OR LOAD
AND LOAD
OUT       D002360.6	// IN BUFFER JOG-
MPOP
AND       M02192	// T)L_2nd_19 R JOG+
OUT       D002360.5	// IN BUFFER JOG+
; L153
LOAD      D001360.0	// IN BUFFER CTRL RDY
AND NOT   D001360.A	// IN BUFFER WARNING
AND NOT   D001360.C	// IN BUFFER SVD ERR
AND NOT   M02193	// T)L_2nd_19 R SERVO ON
AND NOT   M00600	// EMERGENCY ALARM
OUT       D002360.1	// IN BUFFER SERVO ON
; L154
LOAD      M0319C	// L_2nd_19 R Pos HOME >
OUT       D002360.4	// IN BUFFER HOME->
; L155
LOAD NOT  M03190	// L_2nd_19 R Pos.1st IDLE >
AND NOT   M01695	// L_2nd_19 R INITIAL ->
NOT
DMOV      D004900 D002372	// IN BUFFER LEFT °¡¼Ó / IN BUFFER °¡¼Ó
DMOV      D004920 D002374	// IN BUFFER LEFT °¨¼Ó / IN BUFFER °¨¼Ó
DMOV      D004940 D002362	// IN-BUFF ¿ÞÂÊ P&P ÁÖ´ÂÀ§Ä¡ / IN BUFFER ¸ñÇ¥À§Ä¡
DMOV      D004960 D002364	// IN BUFFER LEFT ¼Óµµ / IN BUFFER ¸ñÇ¥¼Óµµ
AND       M01695	// L_2nd_19 R INITIAL ->
DMOV      5000 D002364	// IN BUFFER ¸ñÇ¥¼Óµµ
; L160
LOAD      M03191	// L_2nd_19 R Pos.2nd ROTATE >
DMOV      D004902 D002372	// IN BUFFER RIGHT °¡¼Ó / IN BUFFER °¡¼Ó
DMOV      D004922 D002374	// IN BUFFER RIGHT °¨¼Ó / IN BUFFER °¨¼Ó
DMOV      D004942 D002362	// IN-BUFF ¿À¸¥ÂÊ P&P ÁÖ´ÂÀ§Ä¡ / IN BUFFER ¸ñÇ¥À§Ä¡
DMOV      D004962 D002364	// IN BUFFER RIGHT ¼Óµµ / IN BUFFER ¸ñÇ¥¼Óµµ

